// TIA Portal project "Winda2.2" (V15.1)

(* hardware
DEVICE "S7-1200 station_1"  S7-1200 Station
   slot 0: "Rack_0"  S7-1200 Rack  Rack  V1.0
   slot 1: "PLC_1"  CPU 1212C AC/DC/Rly  6ES7 212-1BD30-0XB0  V2.2
DEVICE "HMI_1"  KTP600 Basic color PN
   slot 0: "HMI_1"  KTP600 Basic color PN  6AV6 647-0AD11-3AX0  12.0.0.0
   slot 1: "HMI_RT_1"  KTP600 Basic color PN  6AV6 647-0AD11-3AX0  12.0.0.0
   slot 5: "HMI_1.IE_CP_1"  PROFINET Interface  12.0.0.0
      slot 1: "PROFINET Interface_1"  PROFINET Interface
         slot 1: "Port_1"  Port
*)

// ===== PLC "PLC_1"  CPU 1212C AC/DC/Rly =====

VAR_GLOBAL   // PLC tag table "Default tag table"
   "Btn_0_floor_out" AT %M0.0 : Bool;
   "Btn_1_floor_out" AT %M0.1 : Bool;
   "Btn_2_floor_out" AT %M0.2 : Bool;
   "Btn_3_floor_out" AT %M0.3 : Bool;
   "Btn_4_floor_out" AT %M0.4 : Bool;
   "Btn_5_floor_out" AT %M0.5 : Bool;
   "Btn_6_floor_out" AT %M0.6 : Bool;
   "Btn_7_floor_out" AT %M0.7 : Bool;
   "Btn_8_floor_out" AT %M1.0 : Bool;
   "Btn_9_floor_out" AT %M1.1 : Bool;
   "Btn_10_floor_out" AT %M1.2 : Bool;
   "Btn_0_floor_in" AT %M1.3 : Bool;
   "Btn_1_floor_in" AT %M1.4 : Bool;
   "Btn_2_floor_in" AT %M1.5 : Bool;
   "Btn_3_floor_in" AT %M1.6 : Bool;
   "Btn_4_floor_in" AT %M1.7 : Bool;
   "Btn_5_floor_in" AT %M2.0 : Bool;
   "Btn_6_floor_in" AT %M2.1 : Bool;
   "Btn_7_floor_in" AT %M2.2 : Bool;
   "Btn_8_floor_in" AT %M2.3 : Bool;
   "Btn_9_floor_in" AT %M2.4 : Bool;
   "Btn_10_floor_in" AT %M2.5 : Bool;
   "Btn_emergency" AT %M2.6 : Bool;
   "Btn_open_door" AT %M2.7 : Bool;
   "Btn_close_door" AT %M3.0 : Bool;
   "DO_open_door" AT %M3.1 : Bool;
   "DO_close_door" AT %M3.2 : Bool;
   "DO_move_lift_up" AT %M3.3 : Bool;
   "DO_move_lift_down" AT %M3.4 : Bool;
   "DO_motor_brake" AT %M3.5 : Bool;
   "MoveTimerIN" AT %M3.6 : Bool;
   "DoorTimerIN" AT %M3.7 : Bool;
   "MoveTimerStoppingIN" AT %M4.0 : Bool;
   "Clock_Byte" AT %MB100 : Byte;
   "Clock_10Hz" AT %M100.0 : Bool;
   "Clock_5Hz" AT %M100.1 : Bool;
   "Clock_2.5Hz" AT %M100.2 : Bool;
   "Clock_2Hz" AT %M100.3 : Bool;
   "Clock_1.25Hz" AT %M100.4 : Bool;
   "Clock_1Hz" AT %M100.5 : Bool;
   "Clock_0.625Hz" AT %M100.6 : Bool;
   "Clock_0.5Hz" AT %M100.7 : Bool;
   "HMIElevatorPosition" AT %MW7 : Int;
   "HMIReq_0" AT %M4.1 : Bool;
   "HMIReq_1" AT %M4.2 : Bool;
   "HMIReq_2" AT %M4.3 : Bool;
   "HMIReq_3" AT %M4.4 : Bool;
   "HMIReq_4" AT %M4.5 : Bool;
   "HMIReq_5" AT %M4.6 : Bool;
   "HMIReq_6" AT %M4.7 : Bool;
   "HMIReq_7" AT %M5.0 : Bool;
   "HMIReq_8" AT %M5.1 : Bool;
   "HMIReq_9" AT %M5.2 : Bool;
   "HMIReq_10" AT %M5.3 : Bool;
   "HMIDoorPosition" AT %MW9 : Int;
   "P1" AT %M5.4 : Bool;
   "P2" AT %M5.5 : Bool;
   "P3" AT %M5.6 : Bool;
   "P4" AT %M5.7 : Bool;
   "P5" AT %M6.0 : Bool;
   "P6" AT %M6.1 : Bool;
   "P7" AT %M6.2 : Bool;
   "P8" AT %M6.3 : Bool;
   "N1" AT %M6.4 : Bool;
END_VAR

VAR_GLOBAL CONSTANT   // PLC tag table "Default tag table"
   "ES_IDLE" : Int := 0;
   "ES_DOOR_OPEN" : Int := 1;
   "ES_MOVING_UP" : Int := 2;
   "ES_MOVING_DOWN" : Int := 3;
   "ES_STOPPING" : Int := 4;
END_VAR

DATA_BLOCK "Elevator"   // DB2
{ S7_Optimized_Access := 'TRUE' }
VERSION : 0.1
   VAR
      Requests : Array[0..10] of Bool;
      state : Int;
      currentFloor : Int;
      targetFloor : Int;
      DoorState : Int := 2;
      DoorTimerPT : Time := T#3ms;
      MoveTimerPT : Time := T#2s;
      MoveTimerStoppingPT : Time := T#4s;
      BeforeEmergancyState : Int;
      DoorTimerWasON : Bool;
      MoveTimerWasON : Bool;
      MoveTimerStoppingWasON : Bool;
      DoorTimerET : Time;
      MoveTimerET : Time;
      MoveTimerStoppingET : Time;
      MotorState : Bool;
   END_VAR
BEGIN
END_DATA_BLOCK

DATA_BLOCK "HMIsim_DB"   // DB5
{ S7_Optimized_Access := 'TRUE' }
VERSION : 0.1
// stored: InstanceOfName HMIsim
"HMIsim"
BEGIN
END_DATA_BLOCK

DATA_BLOCK "UpdateDoorPosition_DB"   // DB6
{ S7_Optimized_Access := 'TRUE' }
VERSION : 0.1
// stored: InstanceOfName UpdateDoorPosition
"UpdateDoorPosition"
BEGIN
END_DATA_BLOCK

// folder: System blocks/Program resources

DATA_BLOCK "DoorTimer"   // DB1
{ S7_Optimized_Access := 'TRUE' }
AUTHOR : Simatic
FAMILY : IEC
NAME : IEC_TMR
VERSION : 1.0
// stored: InstanceOfName IEC_TIMER
"IEC_TIMER"
BEGIN
END_DATA_BLOCK

DATA_BLOCK "MoveTimer"   // DB3
{ S7_Optimized_Access := 'TRUE' }
AUTHOR : Simatic
FAMILY : IEC
NAME : IEC_TMR
VERSION : 1.0
// stored: InstanceOfName IEC_TIMER
"IEC_TIMER"
BEGIN
END_DATA_BLOCK

DATA_BLOCK "MoveTimerStopping"   // DB4
{ S7_Optimized_Access := 'TRUE' }
AUTHOR : Simatic
FAMILY : IEC
NAME : IEC_TMR
VERSION : 1.0
// stored: InstanceOfName IEC_TIMER
"IEC_TIMER"
BEGIN
END_DATA_BLOCK

// folder: (top level)

FUNCTION_BLOCK "HMIsim"   // FB1, LAD
{ S7_Optimized_Access := 'TRUE' }
VERSION : 0.1
   VAR_INPUT
      StartTravel : Bool;
      TargetFloorIndex : Int;
   END_VAR
   VAR_OUTPUT
      ElevatorPos : Int;
   END_VAR
   VAR_TEMP
      direction : Int;
      CurrentStartPos : Int;
      NextFloorPos : Int;
      temp1 : Int;
      ET_int : Int;
      PositionProgress : Real;
      ET_R : Real;
      temp2 : Real;
   END_VAR
   VAR CONSTANT
      StepDistance : Int := 21;
      TotalRange : Int := 210;
      TotalSteps : Int := 10;
   END_VAR
   VAR_TEMP   // added for the SCL form of the ladder/FBD networks
      _w1 : Bool;
      _w2 : Bool;
      _w3 : Bool;
      _w4 : Bool;
   END_VAR
BEGIN

REGION Network 1
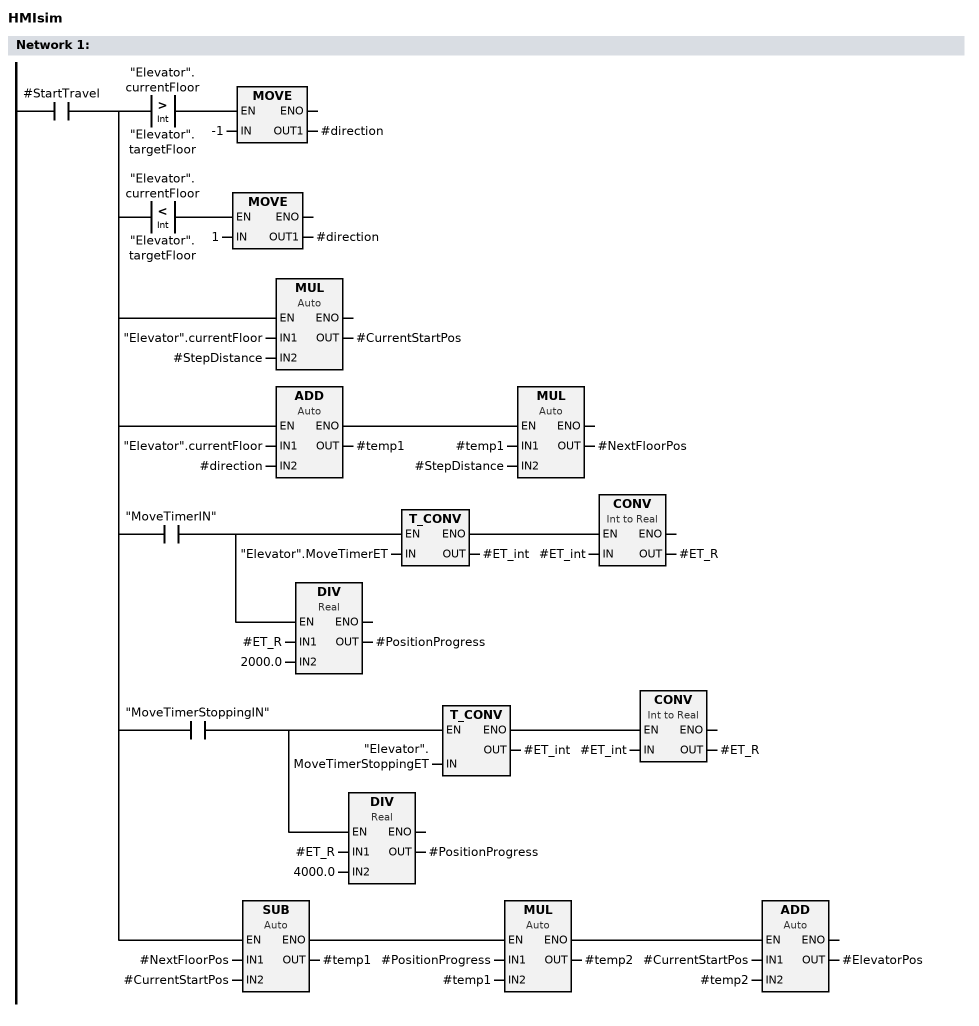
   // ENO of a box is taken as its EN; it also drops when the box reports an error
   IF #StartTravel AND ("Elevator".currentFloor > "Elevator".targetFloor) THEN #direction := -1; END_IF;
   IF #StartTravel AND ("Elevator".currentFloor < "Elevator".targetFloor) THEN #direction := 1; END_IF;
   IF #StartTravel THEN
       #CurrentStartPos := "Elevator".currentFloor * #StepDistance;
       #temp1 := "Elevator".currentFloor + #direction;
       #NextFloorPos := #temp1 * #StepDistance;
   END_IF;
   #_w1 := #StartTravel AND "MoveTimerIN";
   #_w2 := #StartTravel AND "MoveTimerIN";
   IF #_w2 THEN
       #ET_int := T_CONV(IN := "Elevator".MoveTimerET);
       #ET_R := INT_TO_REAL(#ET_int);
   END_IF;
   IF #_w1 THEN #PositionProgress := #ET_R / 2000.0; END_IF;
   #_w3 := #StartTravel AND "MoveTimerStoppingIN";
   #_w4 := #StartTravel AND "MoveTimerStoppingIN";
   IF #_w4 THEN
       #ET_int := T_CONV(IN := "Elevator".MoveTimerStoppingET);
       #ET_R := INT_TO_REAL(#ET_int);
   END_IF;
   IF #_w3 THEN #PositionProgress := #ET_R / 4000.0; END_IF;
   IF #StartTravel THEN
       #temp1 := #NextFloorPos - #CurrentStartPos;
       #temp2 := #PositionProgress * #temp1;
       #ElevatorPos := #CurrentStartPos + #temp2;
   END_IF;
END_REGION
END_FUNCTION_BLOCK

FUNCTION_BLOCK "UpdateDoorPosition"   // FB2, LAD
{ S7_Optimized_Access := 'TRUE' }
VERSION : 0.1
   VAR_INPUT
      TimeElapsed : Time;
   END_VAR
   VAR
      DoorRange : Real := 30.0;
      DoorTimeTotal : Time := T#3s;
   END_VAR
   VAR_TEMP
      TimeFraction : Real;
      Temp_1 : Int;
      Temp_2 : Int;
      Temp_3 : Real;
   END_VAR
BEGIN

REGION Network 1
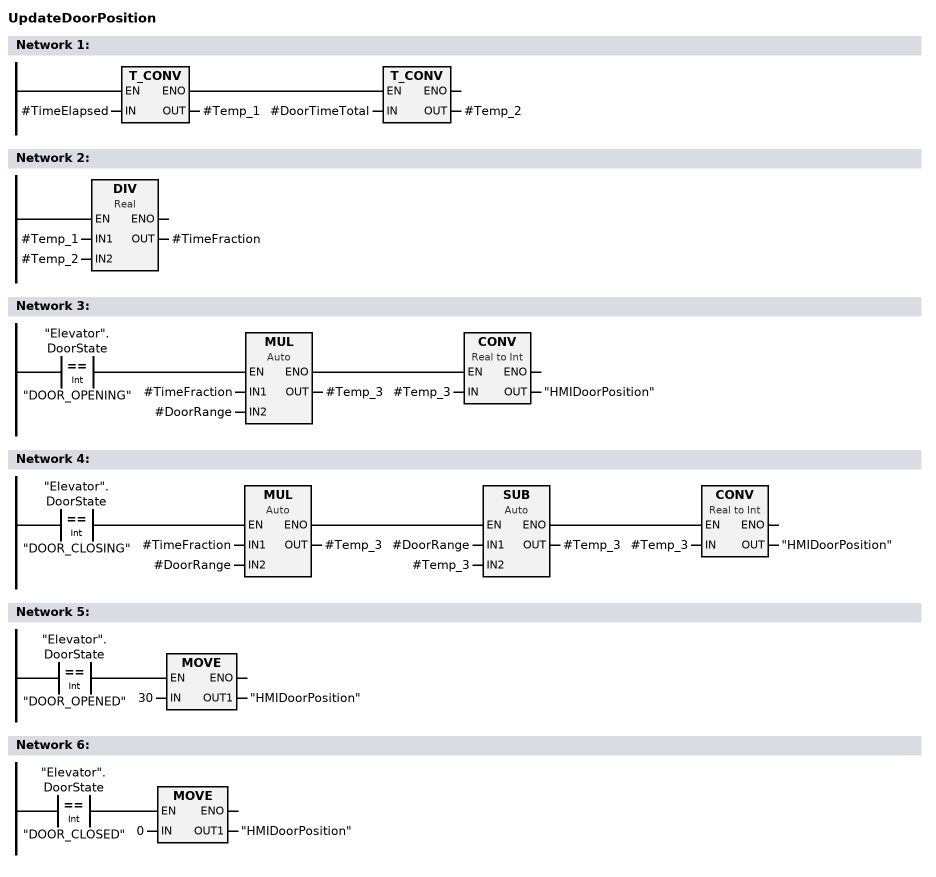
   // ENO of a box is taken as its EN; it also drops when the box reports an error
   #Temp_1 := T_CONV(IN := #TimeElapsed);
   #Temp_2 := T_CONV(IN := #DoorTimeTotal);
END_REGION

REGION Network 2
   RUNG wire#powerrail
      { S7_Templates := "SrcType := Real" } Div(in1 := #Temp_1, in2 := #Temp_2, out => #TimeFraction)
   END_RUNG
   // the same network as SCL:
   #TimeFraction := #Temp_1 / #Temp_2;
END_REGION

REGION Network 3
   RUNG wire#powerrail
      { S7_Templates := "SrcType := Int" } EQ_Contact(in1 := "Elevator".DoorState, in2 := "DOOR_OPENING")
      Mul(in1 := #TimeFraction, in2 := #DoorRange, out => #Temp_3)
      { S7_Templates := "[SrcType := Real, DestType := Int]" } Convert(in := #Temp_3, out => "HMIDoorPosition")
   END_RUNG
   // the same network as SCL:
   IF "Elevator".DoorState = "DOOR_OPENING" THEN
       #Temp_3 := #TimeFraction * #DoorRange;
       "HMIDoorPosition" := REAL_TO_INT(#Temp_3);
   END_IF;
END_REGION

REGION Network 4
   RUNG wire#powerrail
      { S7_Templates := "SrcType := Int" } EQ_Contact(in1 := "Elevator".DoorState, in2 := "DOOR_CLOSING")
      Mul(in1 := #TimeFraction, in2 := #DoorRange, out => #Temp_3)
      Sub(in1 := #DoorRange, in2 := #Temp_3, out => #Temp_3)
      { S7_Templates := "[SrcType := Real, DestType := Int]" } Convert(in := #Temp_3, out => "HMIDoorPosition")
   END_RUNG
   // the same network as SCL:
   IF "Elevator".DoorState = "DOOR_CLOSING" THEN
       #Temp_3 := #TimeFraction * #DoorRange;
       #Temp_3 := #DoorRange - #Temp_3;
       "HMIDoorPosition" := REAL_TO_INT(#Temp_3);
   END_IF;
END_REGION

REGION Network 5
   RUNG wire#powerrail
      { S7_Templates := "SrcType := Int" } EQ_Contact(in1 := "Elevator".DoorState, in2 := "DOOR_OPENED")
      Move(in := 30, out1 => "HMIDoorPosition")
   END_RUNG
   // the same network as SCL:
   IF "Elevator".DoorState = "DOOR_OPENED" THEN "HMIDoorPosition" := 30; END_IF;
END_REGION

REGION Network 6
   RUNG wire#powerrail
      { S7_Templates := "SrcType := Int" } EQ_Contact(in1 := "Elevator".DoorState, in2 := "DOOR_CLOSED")
      Move(in := 0, out1 => "HMIDoorPosition")
   END_RUNG
   // the same network as SCL:
   IF "Elevator".DoorState = "DOOR_CLOSED" THEN "HMIDoorPosition" := 0; END_IF;
END_REGION
END_FUNCTION_BLOCK

FUNCTION "GetPendingRequests" : Void   // FC2, LAD
{ S7_Optimized_Access := 'TRUE' }
VERSION : 0.1
   VAR_INPUT
      Btn_0_floor_out : Bool;
      Btn_1_floor_out : Bool;
      Btn_2_floor_out : Bool;
      Btn_3_floor_out : Bool;
      Btn_4_floor_out : Bool;
      Btn_5_floor_out : Bool;
      Btn_6_floor_out : Bool;
      Btn_7_floor_out : Bool;
      Btn_8_floor_out : Bool;
      Btn_9_floor_out : Bool;
      Btn_10_floor_out : Bool;
      Btn_0_floor_in : Bool;
      Btn_1_floor_in : Bool;
      Btn_2_floor_in : Bool;
      Btn_3_floor_in : Bool;
      Btn_4_floor_in : Bool;
      Btn_5_floor_in : Bool;
      Btn_6_floor_in : Bool;
      Btn_7_floor_in : Bool;
      Btn_8_floor_in : Bool;
      Btn_9_floor_in : Bool;
      Btn_10_floor_in : Bool;
   END_VAR
   VAR_OUTPUT
      requests : Array[0..10] of Bool;
   END_VAR
BEGIN

REGION Network 1
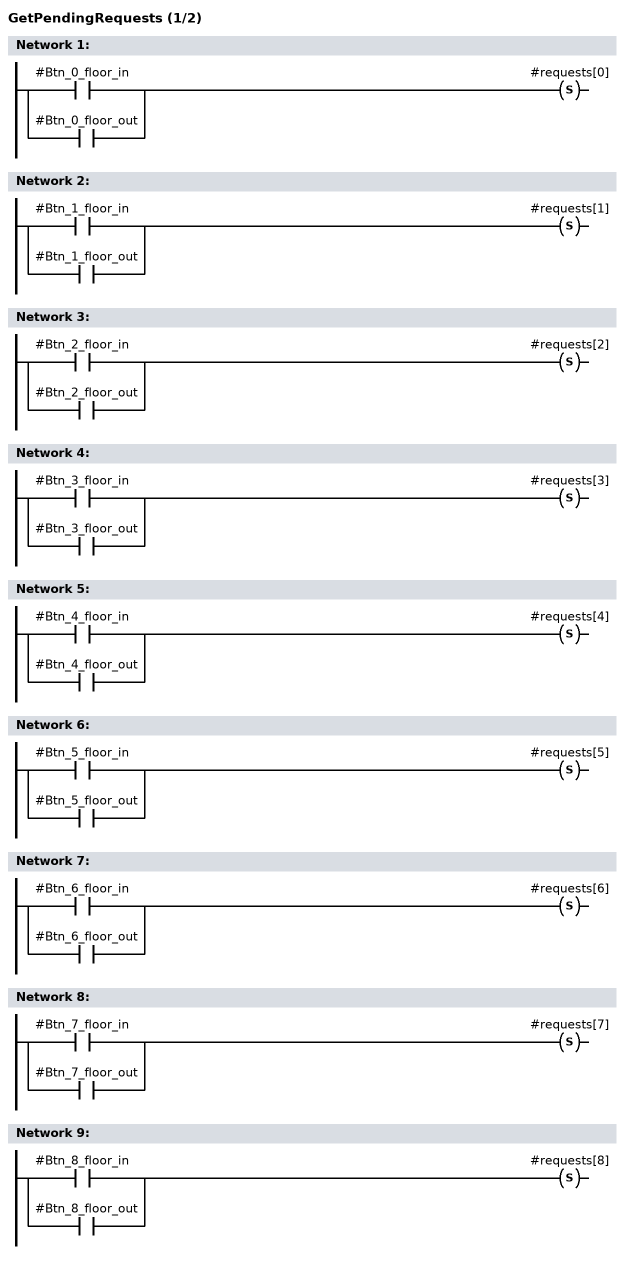
   RUNG wire#powerrail
      Contact( #Btn_0_floor_in )
      wire#w1
      S_Coil( #requests[0] )
   END_RUNG
   RUNG wire#powerrail
      Contact( #Btn_0_floor_out )
   END_RUNG wire#w1
   // the same network as SCL:
   IF #Btn_0_floor_in OR #Btn_0_floor_out THEN #requests[0] := TRUE; END_IF;
END_REGION

REGION Network 2
   RUNG wire#powerrail
      Contact( #Btn_1_floor_in )
      wire#w1
      S_Coil( #requests[1] )
   END_RUNG
   RUNG wire#powerrail
      Contact( #Btn_1_floor_out )
   END_RUNG wire#w1
   // the same network as SCL:
   IF #Btn_1_floor_in OR #Btn_1_floor_out THEN #requests[1] := TRUE; END_IF;
END_REGION

REGION Network 3
   RUNG wire#powerrail
      Contact( #Btn_2_floor_in )
      wire#w1
      S_Coil( #requests[2] )
   END_RUNG
   RUNG wire#powerrail
      Contact( #Btn_2_floor_out )
   END_RUNG wire#w1
   // the same network as SCL:
   IF #Btn_2_floor_in OR #Btn_2_floor_out THEN #requests[2] := TRUE; END_IF;
END_REGION

REGION Network 4
   RUNG wire#powerrail
      Contact( #Btn_3_floor_in )
      wire#w1
      S_Coil( #requests[3] )
   END_RUNG
   RUNG wire#powerrail
      Contact( #Btn_3_floor_out )
   END_RUNG wire#w1
   // the same network as SCL:
   IF #Btn_3_floor_in OR #Btn_3_floor_out THEN #requests[3] := TRUE; END_IF;
END_REGION

REGION Network 5
   RUNG wire#powerrail
      Contact( #Btn_4_floor_in )
      wire#w1
      S_Coil( #requests[4] )
   END_RUNG
   RUNG wire#powerrail
      Contact( #Btn_4_floor_out )
   END_RUNG wire#w1
   // the same network as SCL:
   IF #Btn_4_floor_in OR #Btn_4_floor_out THEN #requests[4] := TRUE; END_IF;
END_REGION

REGION Network 6
   RUNG wire#powerrail
      Contact( #Btn_5_floor_in )
      wire#w1
      S_Coil( #requests[5] )
   END_RUNG
   RUNG wire#powerrail
      Contact( #Btn_5_floor_out )
   END_RUNG wire#w1
   // the same network as SCL:
   IF #Btn_5_floor_in OR #Btn_5_floor_out THEN #requests[5] := TRUE; END_IF;
END_REGION

REGION Network 7
   RUNG wire#powerrail
      Contact( #Btn_6_floor_in )
      wire#w1
      S_Coil( #requests[6] )
   END_RUNG
   RUNG wire#powerrail
      Contact( #Btn_6_floor_out )
   END_RUNG wire#w1
   // the same network as SCL:
   IF #Btn_6_floor_in OR #Btn_6_floor_out THEN #requests[6] := TRUE; END_IF;
END_REGION

REGION Network 8
   RUNG wire#powerrail
      Contact( #Btn_7_floor_in )
      wire#w1
      S_Coil( #requests[7] )
   END_RUNG
   RUNG wire#powerrail
      Contact( #Btn_7_floor_out )
   END_RUNG wire#w1
   // the same network as SCL:
   IF #Btn_7_floor_in OR #Btn_7_floor_out THEN #requests[7] := TRUE; END_IF;
END_REGION

REGION Network 9
   RUNG wire#powerrail
      Contact( #Btn_8_floor_in )
      wire#w1
      S_Coil( #requests[8] )
   END_RUNG
   RUNG wire#powerrail
      Contact( #Btn_8_floor_out )
   END_RUNG wire#w1
   // the same network as SCL:
   IF #Btn_8_floor_in OR #Btn_8_floor_out THEN #requests[8] := TRUE; END_IF;
END_REGION

REGION Network 10
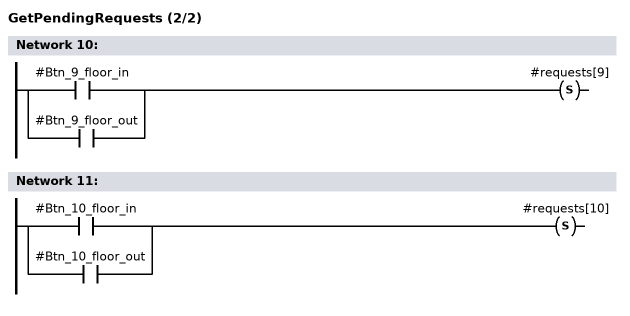
   RUNG wire#powerrail
      Contact( #Btn_9_floor_in )
      wire#w1
      S_Coil( #requests[9] )
   END_RUNG
   RUNG wire#powerrail
      Contact( #Btn_9_floor_out )
   END_RUNG wire#w1
   // the same network as SCL:
   IF #Btn_9_floor_in OR #Btn_9_floor_out THEN #requests[9] := TRUE; END_IF;
END_REGION

REGION Network 11
   RUNG wire#powerrail
      Contact( #Btn_10_floor_in )
      wire#w1
      S_Coil( #requests[10] )
   END_RUNG
   RUNG wire#powerrail
      Contact( #Btn_10_floor_out )
   END_RUNG wire#w1
   // the same network as SCL:
   IF #Btn_10_floor_in OR #Btn_10_floor_out THEN #requests[10] := TRUE; END_IF;
END_REGION
END_FUNCTION

FUNCTION "RequestExists" : Bool   // FC3, LAD
{ S7_Optimized_Access := 'TRUE' }
VERSION : 0.1
BEGIN

REGION Network 1
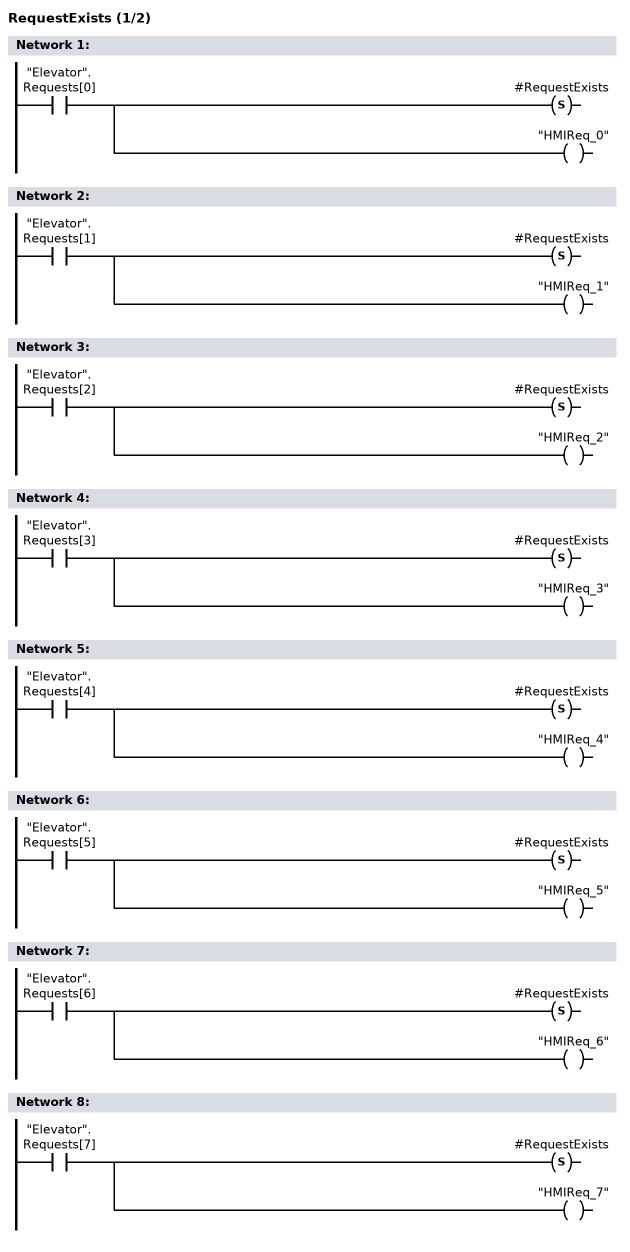
   RUNG wire#powerrail
      Contact( "Elevator".Requests[0] )
      wire#w1
      S_Coil( #RequestExists )
   END_RUNG
   RUNG wire#w1
      Coil( "HMIReq_0" )
   END_RUNG
   // the same network as SCL:
   IF "Elevator".Requests[0] THEN #RequestExists := TRUE; END_IF;
   "HMIReq_0" := "Elevator".Requests[0];
END_REGION

REGION Network 2
   RUNG wire#powerrail
      Contact( "Elevator".Requests[1] )
      wire#w1
      S_Coil( #RequestExists )
   END_RUNG
   RUNG wire#w1
      Coil( "HMIReq_1" )
   END_RUNG
   // the same network as SCL:
   IF "Elevator".Requests[1] THEN #RequestExists := TRUE; END_IF;
   "HMIReq_1" := "Elevator".Requests[1];
END_REGION

REGION Network 3
   RUNG wire#powerrail
      Contact( "Elevator".Requests[2] )
      wire#w1
      S_Coil( #RequestExists )
   END_RUNG
   RUNG wire#w1
      Coil( "HMIReq_2" )
   END_RUNG
   // the same network as SCL:
   IF "Elevator".Requests[2] THEN #RequestExists := TRUE; END_IF;
   "HMIReq_2" := "Elevator".Requests[2];
END_REGION

REGION Network 4
   RUNG wire#powerrail
      Contact( "Elevator".Requests[3] )
      wire#w1
      S_Coil( #RequestExists )
   END_RUNG
   RUNG wire#w1
      Coil( "HMIReq_3" )
   END_RUNG
   // the same network as SCL:
   IF "Elevator".Requests[3] THEN #RequestExists := TRUE; END_IF;
   "HMIReq_3" := "Elevator".Requests[3];
END_REGION

REGION Network 5
   RUNG wire#powerrail
      Contact( "Elevator".Requests[4] )
      wire#w1
      S_Coil( #RequestExists )
   END_RUNG
   RUNG wire#w1
      Coil( "HMIReq_4" )
   END_RUNG
   // the same network as SCL:
   IF "Elevator".Requests[4] THEN #RequestExists := TRUE; END_IF;
   "HMIReq_4" := "Elevator".Requests[4];
END_REGION

REGION Network 6
   RUNG wire#powerrail
      Contact( "Elevator".Requests[5] )
      wire#w1
      S_Coil( #RequestExists )
   END_RUNG
   RUNG wire#w1
      Coil( "HMIReq_5" )
   END_RUNG
   // the same network as SCL:
   IF "Elevator".Requests[5] THEN #RequestExists := TRUE; END_IF;
   "HMIReq_5" := "Elevator".Requests[5];
END_REGION

REGION Network 7
   RUNG wire#powerrail
      Contact( "Elevator".Requests[6] )
      wire#w1
      S_Coil( #RequestExists )
   END_RUNG
   RUNG wire#w1
      Coil( "HMIReq_6" )
   END_RUNG
   // the same network as SCL:
   IF "Elevator".Requests[6] THEN #RequestExists := TRUE; END_IF;
   "HMIReq_6" := "Elevator".Requests[6];
END_REGION

REGION Network 8
   RUNG wire#powerrail
      Contact( "Elevator".Requests[7] )
      wire#w1
      S_Coil( #RequestExists )
   END_RUNG
   RUNG wire#w1
      Coil( "HMIReq_7" )
   END_RUNG
   // the same network as SCL:
   IF "Elevator".Requests[7] THEN #RequestExists := TRUE; END_IF;
   "HMIReq_7" := "Elevator".Requests[7];
END_REGION

REGION Network 9
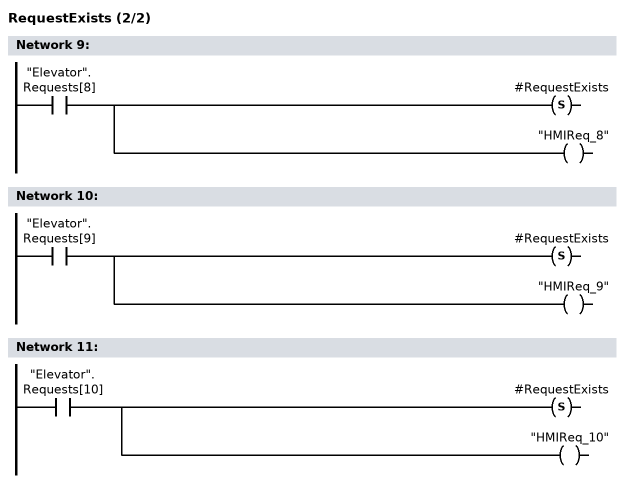
   RUNG wire#powerrail
      Contact( "Elevator".Requests[8] )
      wire#w1
      S_Coil( #RequestExists )
   END_RUNG
   RUNG wire#w1
      Coil( "HMIReq_8" )
   END_RUNG
   // the same network as SCL:
   IF "Elevator".Requests[8] THEN #RequestExists := TRUE; END_IF;
   "HMIReq_8" := "Elevator".Requests[8];
END_REGION

REGION Network 10
   RUNG wire#powerrail
      Contact( "Elevator".Requests[9] )
      wire#w1
      S_Coil( #RequestExists )
   END_RUNG
   RUNG wire#w1
      Coil( "HMIReq_9" )
   END_RUNG
   // the same network as SCL:
   IF "Elevator".Requests[9] THEN #RequestExists := TRUE; END_IF;
   "HMIReq_9" := "Elevator".Requests[9];
END_REGION

REGION Network 11
   RUNG wire#powerrail
      Contact( "Elevator".Requests[10] )
      wire#w1
      S_Coil( #RequestExists )
   END_RUNG
   RUNG wire#w1
      Coil( "HMIReq_10" )
   END_RUNG
   // the same network as SCL:
   IF "Elevator".Requests[10] THEN #RequestExists := TRUE; END_IF;
   "HMIReq_10" := "Elevator".Requests[10];
END_REGION
END_FUNCTION

FUNCTION "GetNextTarget" : Int   // FC4, LAD
{ S7_Optimized_Access := 'TRUE' }
VERSION : 0.1
   VAR_INPUT
      current : Int;
      req : Array[0..10] of Bool;
   END_VAR
   VAR_TEMP
      minDiff : Int;
      diff : Int;
      temp1 : Int;
      temp2 : Int;
      nextTarget : Int;
   END_VAR
   VAR_TEMP   // added for the SCL form of the ladder/FBD networks
      _w1 : Bool;
   END_VAR
BEGIN

REGION Network 1
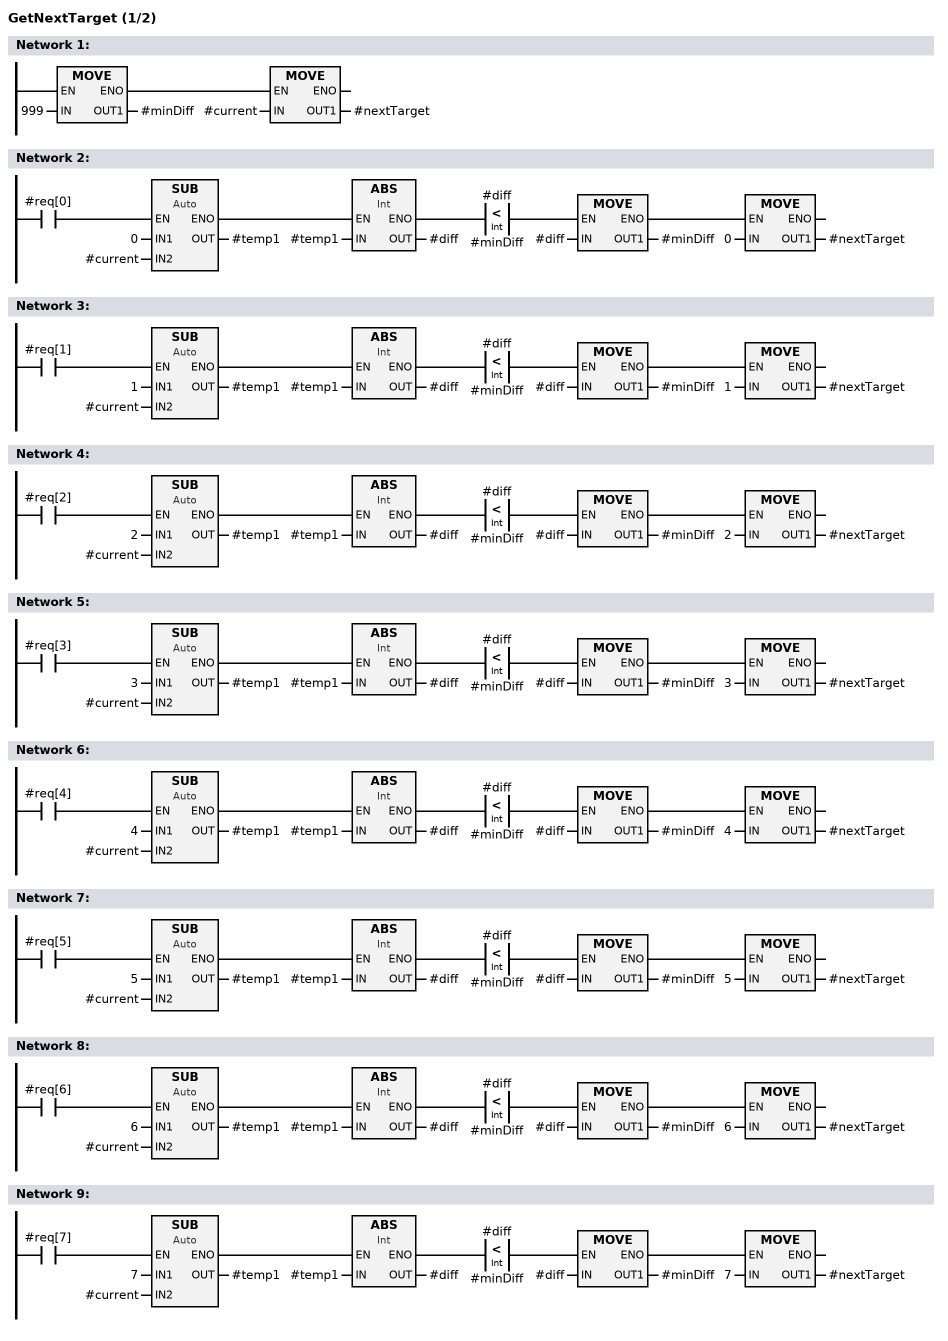
   RUNG wire#powerrail
      { S7_GenerateENO := "TRUE" } Move(in := 999, out1 => #minDiff)
      { S7_GenerateENO := "TRUE" } Move(in := #current, out1 => #nextTarget)
   END_RUNG
   // the same network as SCL:
   // ENO of a box is taken as its EN; it also drops when the box reports an error
   #minDiff := 999;
   #nextTarget := #current;
END_REGION

REGION Network 2
   RUNG wire#powerrail
      Contact( #req[0] )
      { S7_GenerateENO := "TRUE" } Sub(in1 := 0, in2 := #current, out => #temp1)
      { S7_Templates := "SrcType := Int"; S7_GenerateENO := "TRUE" } Abs(in := #temp1, out => #diff)
      { S7_Templates := "SrcType := Int" } LT_Contact(in1 := #diff, in2 := #minDiff)
      { S7_GenerateENO := "TRUE" } Move(in := #diff, out1 => #minDiff)
      { S7_GenerateENO := "TRUE" } Move(in := 0, out1 => #nextTarget)
   END_RUNG
   // the same network as SCL:
   // ENO of a box is taken as its EN; it also drops when the box reports an error
   IF #req[0] THEN
       #temp1 := 0 - #current;
       #diff := ABS(#temp1);
   END_IF;
   #_w1 := #req[0] AND (#diff < #minDiff);
   IF #_w1 THEN
       #minDiff := #diff;
       #nextTarget := 0;
   END_IF;
END_REGION

REGION Network 3
   RUNG wire#powerrail
      Contact( #req[1] )
      { S7_GenerateENO := "TRUE" } Sub(in1 := 1, in2 := #current, out => #temp1)
      { S7_Templates := "SrcType := Int"; S7_GenerateENO := "TRUE" } Abs(in := #temp1, out => #diff)
      { S7_Templates := "SrcType := Int" } LT_Contact(in1 := #diff, in2 := #minDiff)
      { S7_GenerateENO := "TRUE" } Move(in := #diff, out1 => #minDiff)
      { S7_GenerateENO := "TRUE" } Move(in := 1, out1 => #nextTarget)
   END_RUNG
   // the same network as SCL:
   // ENO of a box is taken as its EN; it also drops when the box reports an error
   IF #req[1] THEN
       #temp1 := 1 - #current;
       #diff := ABS(#temp1);
   END_IF;
   #_w1 := #req[1] AND (#diff < #minDiff);
   IF #_w1 THEN
       #minDiff := #diff;
       #nextTarget := 1;
   END_IF;
END_REGION

REGION Network 4
   RUNG wire#powerrail
      Contact( #req[2] )
      { S7_GenerateENO := "TRUE" } Sub(in1 := 2, in2 := #current, out => #temp1)
      { S7_Templates := "SrcType := Int"; S7_GenerateENO := "TRUE" } Abs(in := #temp1, out => #diff)
      { S7_Templates := "SrcType := Int" } LT_Contact(in1 := #diff, in2 := #minDiff)
      { S7_GenerateENO := "TRUE" } Move(in := #diff, out1 => #minDiff)
      { S7_GenerateENO := "TRUE" } Move(in := 2, out1 => #nextTarget)
   END_RUNG
   // the same network as SCL:
   // ENO of a box is taken as its EN; it also drops when the box reports an error
   IF #req[2] THEN
       #temp1 := 2 - #current;
       #diff := ABS(#temp1);
   END_IF;
   #_w1 := #req[2] AND (#diff < #minDiff);
   IF #_w1 THEN
       #minDiff := #diff;
       #nextTarget := 2;
   END_IF;
END_REGION

REGION Network 5
   RUNG wire#powerrail
      Contact( #req[3] )
      { S7_GenerateENO := "TRUE" } Sub(in1 := 3, in2 := #current, out => #temp1)
      { S7_Templates := "SrcType := Int"; S7_GenerateENO := "TRUE" } Abs(in := #temp1, out => #diff)
      { S7_Templates := "SrcType := Int" } LT_Contact(in1 := #diff, in2 := #minDiff)
      { S7_GenerateENO := "TRUE" } Move(in := #diff, out1 => #minDiff)
      { S7_GenerateENO := "TRUE" } Move(in := 3, out1 => #nextTarget)
   END_RUNG
   // the same network as SCL:
   // ENO of a box is taken as its EN; it also drops when the box reports an error
   IF #req[3] THEN
       #temp1 := 3 - #current;
       #diff := ABS(#temp1);
   END_IF;
   #_w1 := #req[3] AND (#diff < #minDiff);
   IF #_w1 THEN
       #minDiff := #diff;
       #nextTarget := 3;
   END_IF;
END_REGION

REGION Network 6
   RUNG wire#powerrail
      Contact( #req[4] )
      { S7_GenerateENO := "TRUE" } Sub(in1 := 4, in2 := #current, out => #temp1)
      { S7_Templates := "SrcType := Int"; S7_GenerateENO := "TRUE" } Abs(in := #temp1, out => #diff)
      { S7_Templates := "SrcType := Int" } LT_Contact(in1 := #diff, in2 := #minDiff)
      { S7_GenerateENO := "TRUE" } Move(in := #diff, out1 => #minDiff)
      { S7_GenerateENO := "TRUE" } Move(in := 4, out1 => #nextTarget)
   END_RUNG
   // the same network as SCL:
   // ENO of a box is taken as its EN; it also drops when the box reports an error
   IF #req[4] THEN
       #temp1 := 4 - #current;
       #diff := ABS(#temp1);
   END_IF;
   #_w1 := #req[4] AND (#diff < #minDiff);
   IF #_w1 THEN
       #minDiff := #diff;
       #nextTarget := 4;
   END_IF;
END_REGION

REGION Network 7
   RUNG wire#powerrail
      Contact( #req[5] )
      { S7_GenerateENO := "TRUE" } Sub(in1 := 5, in2 := #current, out => #temp1)
      { S7_Templates := "SrcType := Int"; S7_GenerateENO := "TRUE" } Abs(in := #temp1, out => #diff)
      { S7_Templates := "SrcType := Int" } LT_Contact(in1 := #diff, in2 := #minDiff)
      { S7_GenerateENO := "TRUE" } Move(in := #diff, out1 => #minDiff)
      { S7_GenerateENO := "TRUE" } Move(in := 5, out1 => #nextTarget)
   END_RUNG
   // the same network as SCL:
   // ENO of a box is taken as its EN; it also drops when the box reports an error
   IF #req[5] THEN
       #temp1 := 5 - #current;
       #diff := ABS(#temp1);
   END_IF;
   #_w1 := #req[5] AND (#diff < #minDiff);
   IF #_w1 THEN
       #minDiff := #diff;
       #nextTarget := 5;
   END_IF;
END_REGION

REGION Network 8
   RUNG wire#powerrail
      Contact( #req[6] )
      { S7_GenerateENO := "TRUE" } Sub(in1 := 6, in2 := #current, out => #temp1)
      { S7_Templates := "SrcType := Int"; S7_GenerateENO := "TRUE" } Abs(in := #temp1, out => #diff)
      { S7_Templates := "SrcType := Int" } LT_Contact(in1 := #diff, in2 := #minDiff)
      { S7_GenerateENO := "TRUE" } Move(in := #diff, out1 => #minDiff)
      { S7_GenerateENO := "TRUE" } Move(in := 6, out1 => #nextTarget)
   END_RUNG
   // the same network as SCL:
   // ENO of a box is taken as its EN; it also drops when the box reports an error
   IF #req[6] THEN
       #temp1 := 6 - #current;
       #diff := ABS(#temp1);
   END_IF;
   #_w1 := #req[6] AND (#diff < #minDiff);
   IF #_w1 THEN
       #minDiff := #diff;
       #nextTarget := 6;
   END_IF;
END_REGION

REGION Network 9
   RUNG wire#powerrail
      Contact( #req[7] )
      { S7_GenerateENO := "TRUE" } Sub(in1 := 7, in2 := #current, out => #temp1)
      { S7_Templates := "SrcType := Int"; S7_GenerateENO := "TRUE" } Abs(in := #temp1, out => #diff)
      { S7_Templates := "SrcType := Int" } LT_Contact(in1 := #diff, in2 := #minDiff)
      { S7_GenerateENO := "TRUE" } Move(in := #diff, out1 => #minDiff)
      { S7_GenerateENO := "TRUE" } Move(in := 7, out1 => #nextTarget)
   END_RUNG
   // the same network as SCL:
   // ENO of a box is taken as its EN; it also drops when the box reports an error
   IF #req[7] THEN
       #temp1 := 7 - #current;
       #diff := ABS(#temp1);
   END_IF;
   #_w1 := #req[7] AND (#diff < #minDiff);
   IF #_w1 THEN
       #minDiff := #diff;
       #nextTarget := 7;
   END_IF;
END_REGION

REGION Network 10
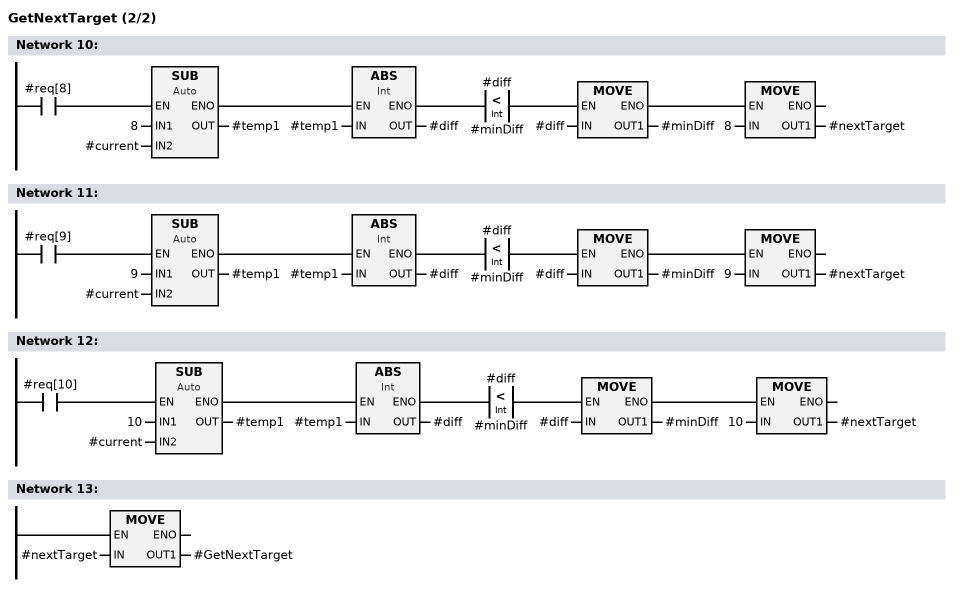
   RUNG wire#powerrail
      Contact( #req[8] )
      { S7_GenerateENO := "TRUE" } Sub(in1 := 8, in2 := #current, out => #temp1)
      { S7_Templates := "SrcType := Int"; S7_GenerateENO := "TRUE" } Abs(in := #temp1, out => #diff)
      { S7_Templates := "SrcType := Int" } LT_Contact(in1 := #diff, in2 := #minDiff)
      { S7_GenerateENO := "TRUE" } Move(in := #diff, out1 => #minDiff)
      { S7_GenerateENO := "TRUE" } Move(in := 8, out1 => #nextTarget)
   END_RUNG
   // the same network as SCL:
   // ENO of a box is taken as its EN; it also drops when the box reports an error
   IF #req[8] THEN
       #temp1 := 8 - #current;
       #diff := ABS(#temp1);
   END_IF;
   #_w1 := #req[8] AND (#diff < #minDiff);
   IF #_w1 THEN
       #minDiff := #diff;
       #nextTarget := 8;
   END_IF;
END_REGION

REGION Network 11
   RUNG wire#powerrail
      Contact( #req[9] )
      { S7_GenerateENO := "TRUE" } Sub(in1 := 9, in2 := #current, out => #temp1)
      { S7_Templates := "SrcType := Int"; S7_GenerateENO := "TRUE" } Abs(in := #temp1, out => #diff)
      { S7_Templates := "SrcType := Int" } LT_Contact(in1 := #diff, in2 := #minDiff)
      { S7_GenerateENO := "TRUE" } Move(in := #diff, out1 => #minDiff)
      { S7_GenerateENO := "TRUE" } Move(in := 9, out1 => #nextTarget)
   END_RUNG
   // the same network as SCL:
   // ENO of a box is taken as its EN; it also drops when the box reports an error
   IF #req[9] THEN
       #temp1 := 9 - #current;
       #diff := ABS(#temp1);
   END_IF;
   #_w1 := #req[9] AND (#diff < #minDiff);
   IF #_w1 THEN
       #minDiff := #diff;
       #nextTarget := 9;
   END_IF;
END_REGION

REGION Network 12
   RUNG wire#powerrail
      Contact( #req[10] )
      { S7_GenerateENO := "TRUE" } Sub(in1 := 10, in2 := #current, out => #temp1)
      { S7_Templates := "SrcType := Int"; S7_GenerateENO := "TRUE" } Abs(in := #temp1, out => #diff)
      { S7_Templates := "SrcType := Int" } LT_Contact(in1 := #diff, in2 := #minDiff)
      { S7_GenerateENO := "TRUE" } Move(in := #diff, out1 => #minDiff)
      { S7_GenerateENO := "TRUE" } Move(in := 10, out1 => #nextTarget)
   END_RUNG
   // the same network as SCL:
   // ENO of a box is taken as its EN; it also drops when the box reports an error
   IF #req[10] THEN
       #temp1 := 10 - #current;
       #diff := ABS(#temp1);
   END_IF;
   #_w1 := #req[10] AND (#diff < #minDiff);
   IF #_w1 THEN
       #minDiff := #diff;
       #nextTarget := 10;
   END_IF;
END_REGION

REGION Network 13
   RUNG wire#powerrail
      { S7_GenerateENO := "TRUE" } Move(in := #nextTarget, out1 => #GetNextTarget)
   END_RUNG
   // the same network as SCL:
   #GetNextTarget := #nextTarget;
END_REGION
END_FUNCTION

ORGANIZATION_BLOCK "Main"   // OB1, LAD, ProgramCycle
TITLE = "Main Program Sweep (Cycle)"
{ S7_Optimized_Access := 'TRUE' }
VERSION : 0.1
   VAR_TEMP
      RET_VAL : Int;
      RET_VAL_1 : Bool;
      flooradded : Bool;
      floorsubtracted : Bool;
      temp1 : Int;
   END_VAR
   VAR_TEMP   // added for the SCL form of the ladder/FBD networks
      _w1 : Bool;
      _w2 : Bool;
      _w3 : Bool;
      _w4 : Bool;
      _w5 : Bool;
      _w6 : Bool;
   END_VAR
BEGIN

REGION Network 1
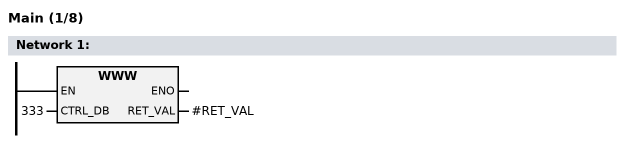
   #RET_VAL := WWW(CTRL_DB := 333);
END_REGION

REGION Network 2
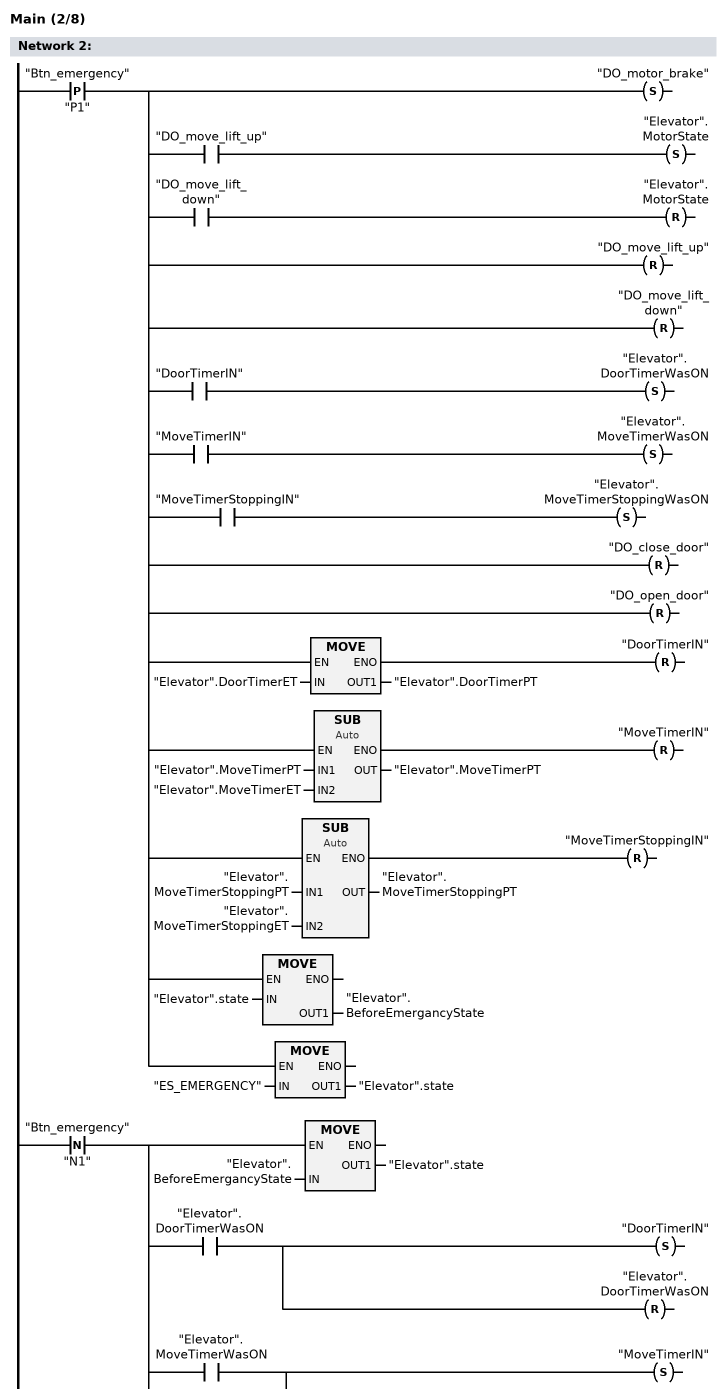
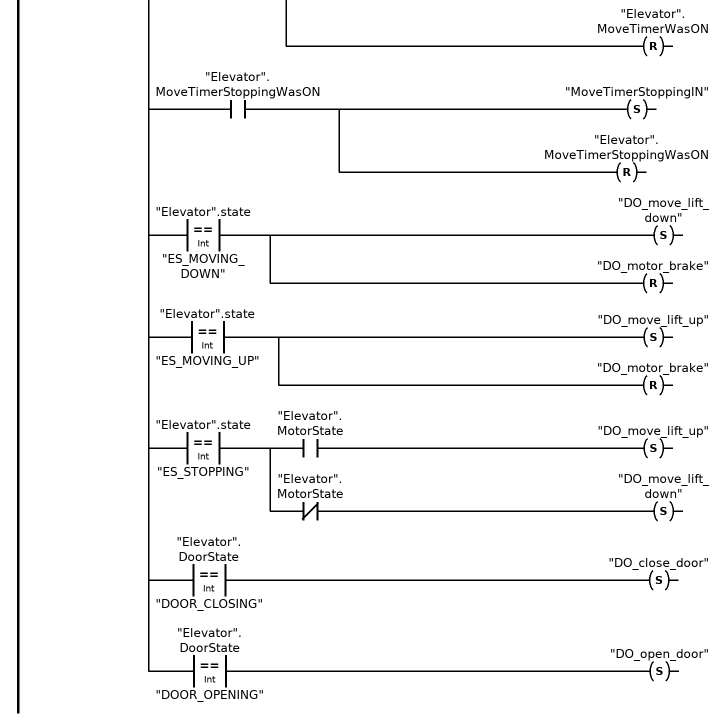
   RUNG wire#powerrail
      P_Contact(operand := "Btn_emergency", bit := "P1")
      wire#w1
      S_Coil( "DO_motor_brake" )
   END_RUNG
   RUNG wire#w1
      Contact( "DO_move_lift_up" )
      S_Coil( "Elevator".MotorState )
   END_RUNG
   RUNG wire#w1
      Contact( "DO_move_lift_down" )
      R_Coil( "Elevator".MotorState )
   END_RUNG
   RUNG wire#w1
      R_Coil( "DO_move_lift_up" )
   END_RUNG
   RUNG wire#w1
      R_Coil( "DO_move_lift_down" )
   END_RUNG
   RUNG wire#w1
      Contact( "DoorTimerIN" )
      S_Coil( "Elevator".DoorTimerWasON )
   END_RUNG
   RUNG wire#w1
      Contact( "MoveTimerIN" )
      S_Coil( "Elevator".MoveTimerWasON )
   END_RUNG
   RUNG wire#w1
      Contact( "MoveTimerStoppingIN" )
      S_Coil( "Elevator".MoveTimerStoppingWasON )
   END_RUNG
   RUNG wire#w1
      R_Coil( "DO_close_door" )
   END_RUNG
   RUNG wire#w1
      R_Coil( "DO_open_door" )
   END_RUNG
   RUNG wire#w1
      Move(in := "Elevator".DoorTimerET, out1 => "Elevator".DoorTimerPT)
      R_Coil( "DoorTimerIN" )
   END_RUNG
   RUNG wire#w1
      Sub(in1 := "Elevator".MoveTimerPT, in2 := "Elevator".MoveTimerET, out => "Elevator".MoveTimerPT)
      R_Coil( "MoveTimerIN" )
   END_RUNG
   RUNG wire#w1
      Sub(in1 := "Elevator".MoveTimerStoppingPT, in2 := "Elevator".MoveTimerStoppingET, out => "Elevator".MoveTimerStoppingPT)
      R_Coil( "MoveTimerStoppingIN" )
   END_RUNG
   RUNG wire#w1
      Move(in := "Elevator".state, out1 => "Elevator".BeforeEmergancyState)
   END_RUNG
   RUNG wire#w1
      Move(in := "ES_EMERGENCY", out1 => "Elevator".state)
   END_RUNG
   RUNG wire#powerrail
      N_Contact(operand := "Btn_emergency", bit := "N1")
      wire#w2
      Move(in := "Elevator".BeforeEmergancyState, out1 => "Elevator".state)
   END_RUNG
   RUNG wire#w2
      Contact( "Elevator".DoorTimerWasON )
      wire#w3
      S_Coil( "DoorTimerIN" )
   END_RUNG
   RUNG wire#w3
      R_Coil( "Elevator".DoorTimerWasON )
   END_RUNG
   RUNG wire#w2
      Contact( "Elevator".MoveTimerWasON )
      wire#w4
      S_Coil( "MoveTimerIN" )
   END_RUNG
   RUNG wire#w4
      R_Coil( "Elevator".MoveTimerWasON )
   END_RUNG
   RUNG wire#w2
      Contact( "Elevator".MoveTimerStoppingWasON )
      wire#w5
      S_Coil( "MoveTimerStoppingIN" )
   END_RUNG
   RUNG wire#w5
      R_Coil( "Elevator".MoveTimerStoppingWasON )
   END_RUNG
   RUNG wire#w2
      { S7_Templates := "SrcType := Int" } EQ_Contact(in1 := "Elevator".state, in2 := "ES_MOVING_DOWN")
      wire#w6
      S_Coil( "DO_move_lift_down" )
   END_RUNG
   RUNG wire#w6
      R_Coil( "DO_motor_brake" )
   END_RUNG
   RUNG wire#w2
      { S7_Templates := "SrcType := Int" } EQ_Contact(in1 := "Elevator".state, in2 := "ES_MOVING_UP")
      wire#w7
      S_Coil( "DO_move_lift_up" )
   END_RUNG
   RUNG wire#w7
      R_Coil( "DO_motor_brake" )
   END_RUNG
   RUNG wire#w2
      { S7_Templates := "SrcType := Int" } EQ_Contact(in1 := "Elevator".state, in2 := "ES_STOPPING")
      wire#w8
      Contact( "Elevator".MotorState )
      S_Coil( "DO_move_lift_up" )
   END_RUNG
   RUNG wire#w8
      I_Contact( "Elevator".MotorState )
      S_Coil( "DO_move_lift_down" )
   END_RUNG
   RUNG wire#w2
      { S7_Templates := "SrcType := Int" } EQ_Contact(in1 := "Elevator".DoorState, in2 := "DOOR_CLOSING")
      S_Coil( "DO_close_door" )
   END_RUNG
   RUNG wire#w2
      { S7_Templates := "SrcType := Int" } EQ_Contact(in1 := "Elevator".DoorState, in2 := "DOOR_OPENING")
      S_Coil( "DO_open_door" )
   END_RUNG
   // the same network as SCL:
   #_w1 := "Btn_emergency" AND NOT "P1";   // rising edge of "Btn_emergency"
   "P1" := "Btn_emergency";
   IF #_w1 THEN "DO_motor_brake" := TRUE; END_IF;
   IF #_w1 AND "DO_move_lift_up" THEN "Elevator".MotorState := TRUE; END_IF;
   IF #_w1 AND "DO_move_lift_down" THEN "Elevator".MotorState := FALSE; END_IF;
   IF #_w1 THEN
       "DO_move_lift_up" := FALSE;
       "DO_move_lift_down" := FALSE;
   END_IF;
   IF #_w1 AND "DoorTimerIN" THEN "Elevator".DoorTimerWasON := TRUE; END_IF;
   IF #_w1 AND "MoveTimerIN" THEN "Elevator".MoveTimerWasON := TRUE; END_IF;
   IF #_w1 AND "MoveTimerStoppingIN" THEN "Elevator".MoveTimerStoppingWasON := TRUE; END_IF;
   IF #_w1 THEN
       "DO_close_door" := FALSE;
       "DO_open_door" := FALSE;
       "Elevator".DoorTimerPT := "Elevator".DoorTimerET;
       "DoorTimerIN" := FALSE;
       "Elevator".MoveTimerPT := "Elevator".MoveTimerPT - "Elevator".MoveTimerET;
       "MoveTimerIN" := FALSE;
       "Elevator".MoveTimerStoppingPT := "Elevator".MoveTimerStoppingPT - "Elevator".MoveTimerStoppingET;
       "MoveTimerStoppingIN" := FALSE;
       "Elevator".BeforeEmergancyState := "Elevator".state;
       "Elevator".state := "ES_EMERGENCY";
   END_IF;
   #_w2 := NOT "Btn_emergency" AND "N1";   // falling edge of "Btn_emergency"
   "N1" := "Btn_emergency";
   IF #_w2 THEN "Elevator".state := "Elevator".BeforeEmergancyState; END_IF;
   IF #_w2 AND "Elevator".DoorTimerWasON THEN
       "DoorTimerIN" := TRUE;
       "Elevator".DoorTimerWasON := FALSE;
   END_IF;
   IF #_w2 AND "Elevator".MoveTimerWasON THEN
       "MoveTimerIN" := TRUE;
       "Elevator".MoveTimerWasON := FALSE;
   END_IF;
   IF #_w2 AND "Elevator".MoveTimerStoppingWasON THEN
       "MoveTimerStoppingIN" := TRUE;
       "Elevator".MoveTimerStoppingWasON := FALSE;
   END_IF;
   IF #_w2 AND ("Elevator".state = "ES_MOVING_DOWN") THEN
       "DO_move_lift_down" := TRUE;
       "DO_motor_brake" := FALSE;
   END_IF;
   IF #_w2 AND ("Elevator".state = "ES_MOVING_UP") THEN
       "DO_move_lift_up" := TRUE;
       "DO_motor_brake" := FALSE;
   END_IF;
   #_w3 := #_w2 AND ("Elevator".state = "ES_STOPPING");
   IF #_w3 AND "Elevator".MotorState THEN "DO_move_lift_up" := TRUE; END_IF;
   IF #_w3 AND NOT "Elevator".MotorState THEN "DO_move_lift_down" := TRUE; END_IF;
   IF #_w2 AND ("Elevator".DoorState = "DOOR_CLOSING") THEN "DO_close_door" := TRUE; END_IF;
   IF #_w2 AND ("Elevator".DoorState = "DOOR_OPENING") THEN "DO_open_door" := TRUE; END_IF;
END_REGION

REGION Network 3
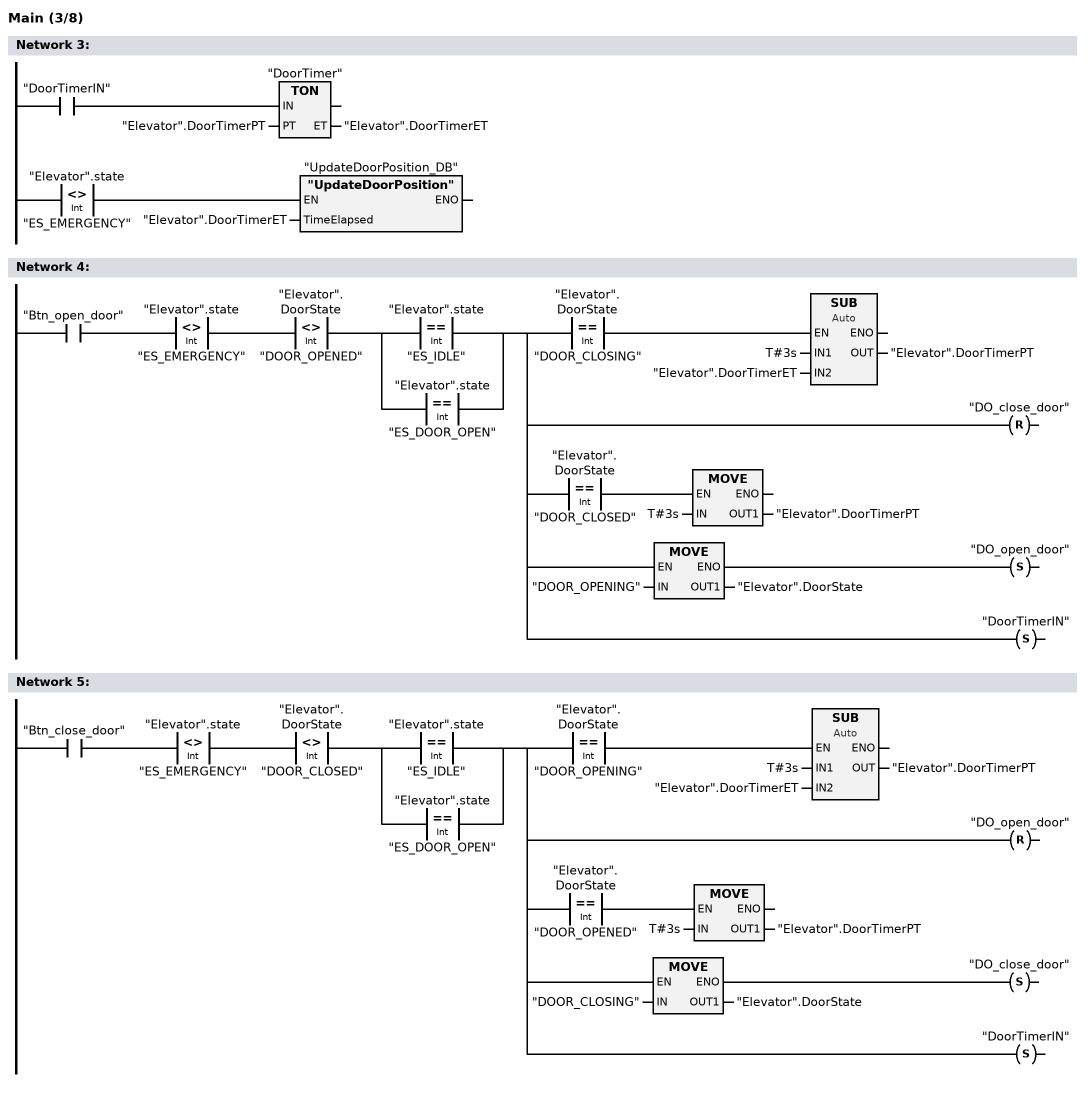
   "DoorTimer".TON(IN := "DoorTimerIN", PT := "Elevator".DoorTimerPT, ET => "Elevator".DoorTimerET);
   IF "Elevator".state <> "ES_EMERGENCY" THEN
       "UpdateDoorPosition_DB"(TimeElapsed := "Elevator".DoorTimerET);   // "UpdateDoorPosition"
   END_IF;
END_REGION

REGION Network 4
   RUNG wire#powerrail
      Contact( "Btn_open_door" )
      { S7_Templates := "SrcType := Int" } NE_Contact(in1 := "Elevator".state, in2 := "ES_EMERGENCY")
      { S7_Templates := "SrcType := Int" } NE_Contact(in1 := "Elevator".DoorState, in2 := "DOOR_OPENED")
      wire#w1
      { S7_Templates := "SrcType := Int" } EQ_Contact(in1 := "Elevator".state, in2 := "ES_IDLE")
      wire#w2
      { S7_Templates := "SrcType := Int" } EQ_Contact(in1 := "Elevator".DoorState, in2 := "DOOR_CLOSING")
      Sub(in1 := T#3s, in2 := "Elevator".DoorTimerET, out => "Elevator".DoorTimerPT)
   END_RUNG
   RUNG wire#w1
      { S7_Templates := "SrcType := Int" } EQ_Contact(in1 := "Elevator".state, in2 := "ES_DOOR_OPEN")
   END_RUNG wire#w2
   RUNG wire#w2
      R_Coil( "DO_close_door" )
   END_RUNG
   RUNG wire#w2
      { S7_Templates := "SrcType := Int" } EQ_Contact(in1 := "Elevator".DoorState, in2 := "DOOR_CLOSED")
      Move(in := T#3s, out1 => "Elevator".DoorTimerPT)
   END_RUNG
   RUNG wire#w2
      Move(in := "DOOR_OPENING", out1 => "Elevator".DoorState)
      S_Coil( "DO_open_door" )
   END_RUNG
   RUNG wire#w2
      S_Coil( "DoorTimerIN" )
   END_RUNG
   // the same network as SCL:
   #_w1 := "Btn_open_door" AND ("Elevator".state <> "ES_EMERGENCY") AND ("Elevator".DoorState <> "DOOR_OPENED") AND (("Elevator".state = "ES_IDLE") OR ("Elevator".state = "ES_DOOR_OPEN"));
   IF #_w1 AND ("Elevator".DoorState = "DOOR_CLOSING") THEN
       "Elevator".DoorTimerPT := T#3s - "Elevator".DoorTimerET;
   END_IF;
   IF #_w1 THEN "DO_close_door" := FALSE; END_IF;
   IF #_w1 AND ("Elevator".DoorState = "DOOR_CLOSED") THEN "Elevator".DoorTimerPT := T#3s; END_IF;
   IF #_w1 THEN
       "Elevator".DoorState := "DOOR_OPENING";
       "DO_open_door" := TRUE;
       "DoorTimerIN" := TRUE;
   END_IF;
END_REGION

REGION Network 5
   RUNG wire#powerrail
      Contact( "Btn_close_door" )
      { S7_Templates := "SrcType := Int" } NE_Contact(in1 := "Elevator".state, in2 := "ES_EMERGENCY")
      { S7_Templates := "SrcType := Int" } NE_Contact(in1 := "Elevator".DoorState, in2 := "DOOR_CLOSED")
      wire#w1
      { S7_Templates := "SrcType := Int" } EQ_Contact(in1 := "Elevator".state, in2 := "ES_IDLE")
      wire#w2
      { S7_Templates := "SrcType := Int" } EQ_Contact(in1 := "Elevator".DoorState, in2 := "DOOR_OPENING")
      Sub(in1 := T#3s, in2 := "Elevator".DoorTimerET, out => "Elevator".DoorTimerPT)
   END_RUNG
   RUNG wire#w1
      { S7_Templates := "SrcType := Int" } EQ_Contact(in1 := "Elevator".state, in2 := "ES_DOOR_OPEN")
   END_RUNG wire#w2
   RUNG wire#w2
      R_Coil( "DO_open_door" )
   END_RUNG
   RUNG wire#w2
      { S7_Templates := "SrcType := Int" } EQ_Contact(in1 := "Elevator".DoorState, in2 := "DOOR_OPENED")
      Move(in := T#3s, out1 => "Elevator".DoorTimerPT)
   END_RUNG
   RUNG wire#w2
      Move(in := "DOOR_CLOSING", out1 => "Elevator".DoorState)
      S_Coil( "DO_close_door" )
   END_RUNG
   RUNG wire#w2
      S_Coil( "DoorTimerIN" )
   END_RUNG
   // the same network as SCL:
   #_w1 := "Btn_close_door" AND ("Elevator".state <> "ES_EMERGENCY") AND ("Elevator".DoorState <> "DOOR_CLOSED") AND (("Elevator".state = "ES_IDLE") OR ("Elevator".state = "ES_DOOR_OPEN"));
   IF #_w1 AND ("Elevator".DoorState = "DOOR_OPENING") THEN
       "Elevator".DoorTimerPT := T#3s - "Elevator".DoorTimerET;
   END_IF;
   IF #_w1 THEN "DO_open_door" := FALSE; END_IF;
   IF #_w1 AND ("Elevator".DoorState = "DOOR_OPENED") THEN "Elevator".DoorTimerPT := T#3s; END_IF;
   IF #_w1 THEN
       "Elevator".DoorState := "DOOR_CLOSING";
       "DO_close_door" := TRUE;
       "DoorTimerIN" := TRUE;
   END_IF;
END_REGION

REGION Network 6
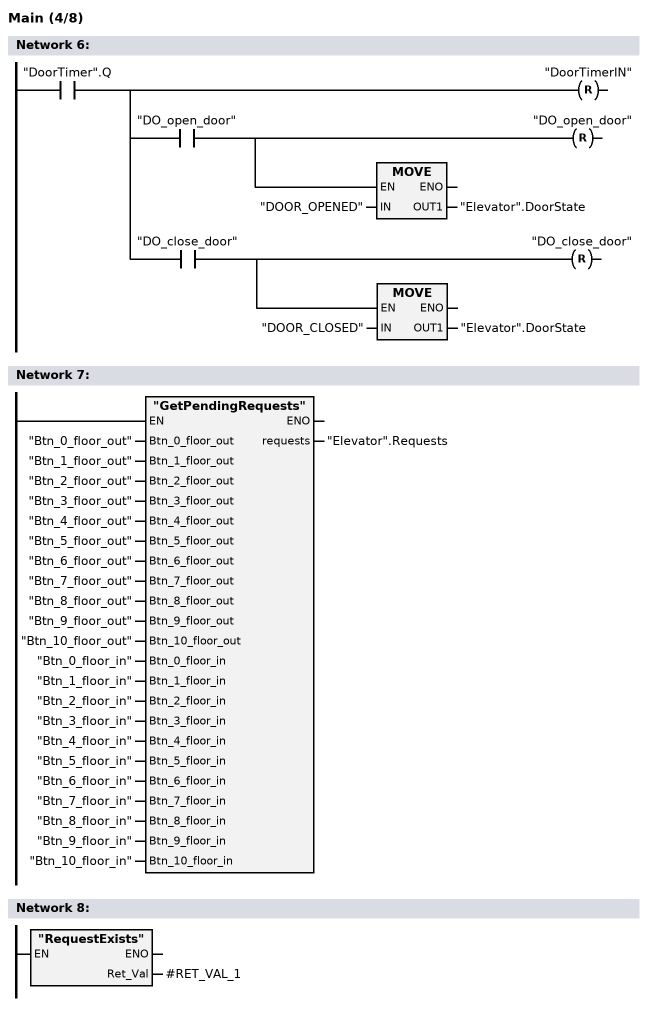
   RUNG wire#powerrail
      Contact( "DoorTimer".Q )
      wire#w1
      R_Coil( "DoorTimerIN" )
   END_RUNG
   RUNG wire#w1
      Contact( "DO_open_door" )
      wire#w2
      R_Coil( "DO_open_door" )
   END_RUNG
   RUNG wire#w2
      Move(in := "DOOR_OPENED", out1 => "Elevator".DoorState)
   END_RUNG
   RUNG wire#w1
      Contact( "DO_close_door" )
      wire#w3
      R_Coil( "DO_close_door" )
   END_RUNG
   RUNG wire#w3
      Move(in := "DOOR_CLOSED", out1 => "Elevator".DoorState)
   END_RUNG
   // the same network as SCL:
   IF "DoorTimer".Q THEN "DoorTimerIN" := FALSE; END_IF;
   #_w1 := "DoorTimer".Q AND "DO_open_door";
   IF #_w1 THEN
       "DO_open_door" := FALSE;
       "Elevator".DoorState := "DOOR_OPENED";
   END_IF;
   #_w2 := "DoorTimer".Q AND "DO_close_door";
   IF #_w2 THEN
       "DO_close_door" := FALSE;
       "Elevator".DoorState := "DOOR_CLOSED";
   END_IF;
END_REGION

REGION Network 7
   RUNG wire#powerrail
      "GetPendingRequests"(Btn_0_floor_out := "Btn_0_floor_out", Btn_1_floor_out := "Btn_1_floor_out", Btn_2_floor_out := "Btn_2_floor_out", Btn_3_floor_out := "Btn_3_floor_out", Btn_4_floor_out := "Btn_4_floor_out", Btn_5_floor_out := "Btn_5_floor_out", Btn_6_floor_out := "Btn_6_floor_out", Btn_7_floor_out := "Btn_7_floor_out", Btn_8_floor_out := "Btn_8_floor_out", Btn_9_floor_out := "Btn_9_floor_out", Btn_10_floor_out := "Btn_10_floor_out", Btn_0_floor_in := "Btn_0_floor_in", Btn_1_floor_in := "Btn_1_floor_in", Btn_2_floor_in := "Btn_2_floor_in", Btn_3_floor_in := "Btn_3_floor_in", Btn_4_floor_in := "Btn_4_floor_in", Btn_5_floor_in := "Btn_5_floor_in", Btn_6_floor_in := "Btn_6_floor_in", Btn_7_floor_in := "Btn_7_floor_in", Btn_8_floor_in := "Btn_8_floor_in", Btn_9_floor_in := "Btn_9_floor_in", Btn_10_floor_in := "Btn_10_floor_in", requests => "Elevator".Requests)
   END_RUNG
   // the same network as SCL:
   "GetPendingRequests"(Btn_0_floor_out := "Btn_0_floor_out",
                        Btn_1_floor_out := "Btn_1_floor_out",
                        Btn_2_floor_out := "Btn_2_floor_out",
                        Btn_3_floor_out := "Btn_3_floor_out",
                        Btn_4_floor_out := "Btn_4_floor_out",
                        Btn_5_floor_out := "Btn_5_floor_out",
                        Btn_6_floor_out := "Btn_6_floor_out",
                        Btn_7_floor_out := "Btn_7_floor_out",
                        Btn_8_floor_out := "Btn_8_floor_out",
                        Btn_9_floor_out := "Btn_9_floor_out",
                        Btn_10_floor_out := "Btn_10_floor_out",
                        Btn_0_floor_in := "Btn_0_floor_in",
                        Btn_1_floor_in := "Btn_1_floor_in",
                        Btn_2_floor_in := "Btn_2_floor_in",
                        Btn_3_floor_in := "Btn_3_floor_in",
                        Btn_4_floor_in := "Btn_4_floor_in",
                        Btn_5_floor_in := "Btn_5_floor_in",
                        Btn_6_floor_in := "Btn_6_floor_in",
                        Btn_7_floor_in := "Btn_7_floor_in",
                        Btn_8_floor_in := "Btn_8_floor_in",
                        Btn_9_floor_in := "Btn_9_floor_in",
                        Btn_10_floor_in := "Btn_10_floor_in",
                        requests => "Elevator".Requests);
END_REGION

REGION Network 8
   RUNG wire#powerrail
      "RequestExists"(Ret_Val => #RET_VAL_1)
   END_RUNG
   // the same network as SCL:
   #RET_VAL_1 := "RequestExists"();
END_REGION

REGION Network 9
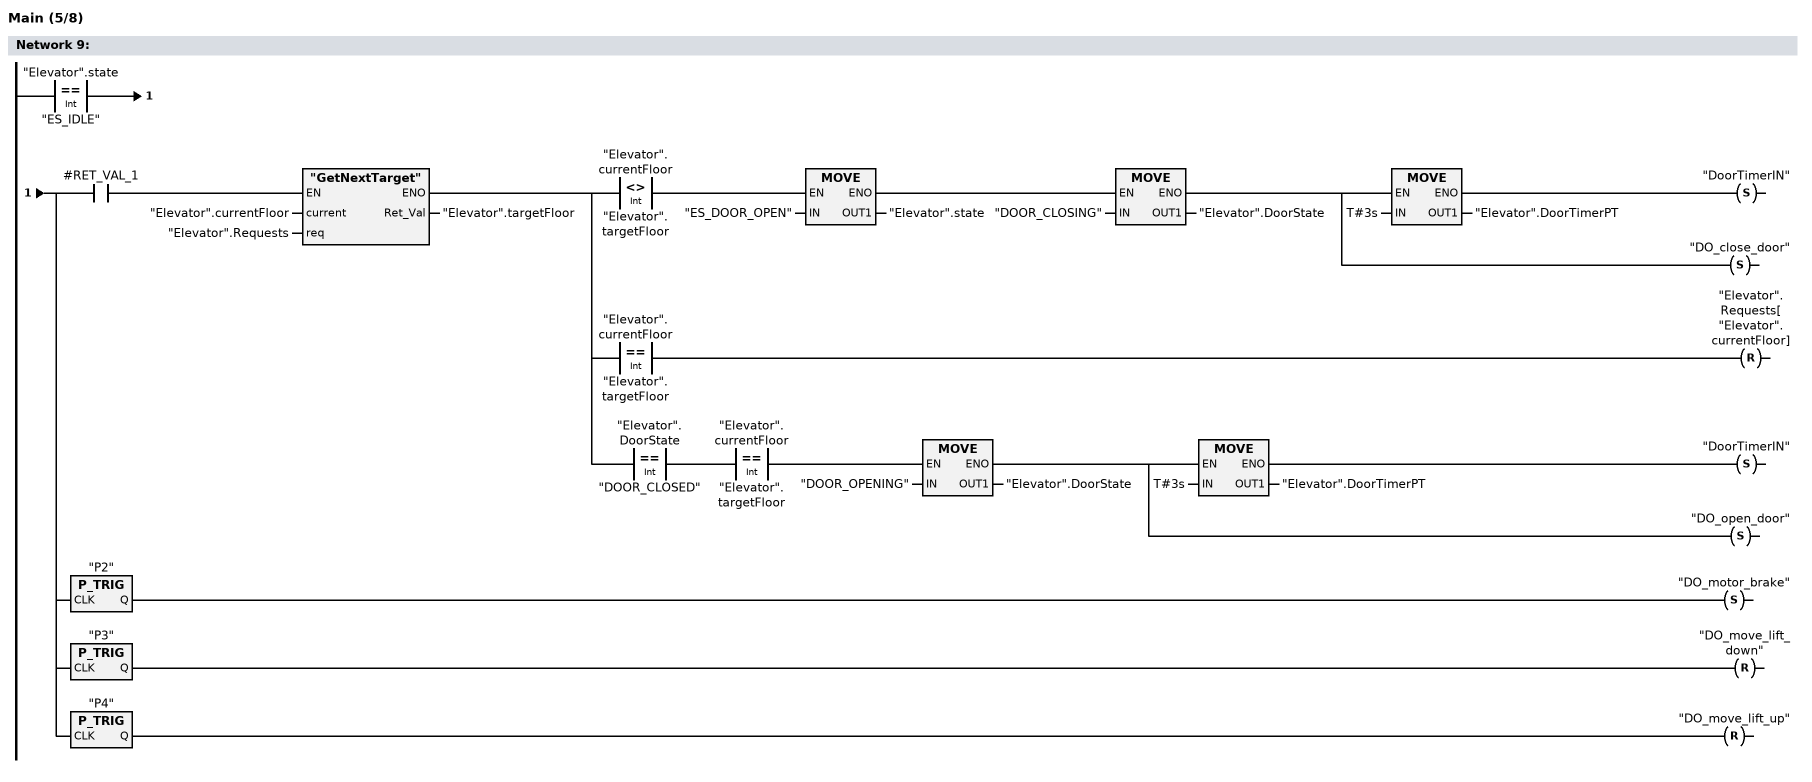
   RUNG wire#powerrail
      { S7_Templates := "SrcType := Int" } EQ_Contact(in1 := "Elevator".state, in2 := "ES_IDLE")
      wire#w1
      Contact( #RET_VAL_1 )
      "GetNextTarget"(current := "Elevator".currentFloor, req := "Elevator".Requests, Ret_Val => "Elevator".targetFloor)
      wire#w2
      { S7_Templates := "SrcType := Int" } NE_Contact(in1 := "Elevator".currentFloor, in2 := "Elevator".targetFloor)
      { S7_GenerateENO := "TRUE" } Move(in := "ES_DOOR_OPEN", out1 => "Elevator".state)
      { S7_GenerateENO := "TRUE" } Move(in := "DOOR_CLOSING", out1 => "Elevator".DoorState)
      wire#w3
      { S7_GenerateENO := "TRUE" } Move(in := T#3s, out1 => "Elevator".DoorTimerPT)
      S_Coil( "DoorTimerIN" )
   END_RUNG
   RUNG wire#w3
      S_Coil( "DO_close_door" )
   END_RUNG
   RUNG wire#w2
      { S7_Templates := "SrcType := Int" } EQ_Contact(in1 := "Elevator".currentFloor, in2 := "Elevator".targetFloor)
      R_Coil( "Elevator".Requests["Elevator".currentFloor] )
   END_RUNG
   RUNG wire#w2
      { S7_Templates := "SrcType := Int" } EQ_Contact(in1 := "Elevator".DoorState, in2 := "DOOR_CLOSED")
      { S7_Templates := "SrcType := Int" } EQ_Contact(in1 := "Elevator".currentFloor, in2 := "Elevator".targetFloor)
      { S7_GenerateENO := "TRUE" } Move(in := "DOOR_OPENING", out1 => "Elevator".DoorState)
      wire#w4
      { S7_GenerateENO := "TRUE" } Move(in := T#3s, out1 => "Elevator".DoorTimerPT)
      S_Coil( "DoorTimerIN" )
   END_RUNG
   RUNG wire#w4
      S_Coil( "DO_open_door" )
   END_RUNG
   RUNG wire#w1
      P_Trig( "P2" )
      S_Coil( "DO_motor_brake" )
   END_RUNG
   RUNG wire#w1
      P_Trig( "P3" )
      R_Coil( "DO_move_lift_down" )
   END_RUNG
   RUNG wire#w1
      P_Trig( "P4" )
      R_Coil( "DO_move_lift_up" )
   END_RUNG
   // the same network as SCL:
   // ENO of a box is taken as its EN; it also drops when the box reports an error
   #_w1 := "Elevator".state = "ES_IDLE";
   "Elevator".targetFloor := "GetNextTarget"(EN := #_w1 AND #RET_VAL_1,
                           current := "Elevator".currentFloor,
                           req := "Elevator".Requests,
                           ENO => #_w2);
   IF #_w2 AND ("Elevator".currentFloor <> "Elevator".targetFloor) THEN
       "Elevator".state := "ES_DOOR_OPEN";
       "Elevator".DoorState := "DOOR_CLOSING";
       "Elevator".DoorTimerPT := T#3s;
       "DoorTimerIN" := TRUE;
       "DO_close_door" := TRUE;
   END_IF;
   IF #_w2 AND ("Elevator".currentFloor = "Elevator".targetFloor) THEN
       "Elevator".Requests["Elevator".currentFloor] := FALSE;
   END_IF;
   #_w3 := #_w2 AND ("Elevator".DoorState = "DOOR_CLOSED") AND ("Elevator".currentFloor = "Elevator".targetFloor);
   IF #_w3 THEN
       "Elevator".DoorState := "DOOR_OPENING";
       "Elevator".DoorTimerPT := T#3s;
       "DoorTimerIN" := TRUE;
       "DO_open_door" := TRUE;
   END_IF;
   #_w4 := #_w1 AND NOT "P2";   // rising edge
   "P2" := #_w1;
   IF #_w4 THEN "DO_motor_brake" := TRUE; END_IF;
   #_w5 := #_w1 AND NOT "P3";   // rising edge
   "P3" := #_w1;
   IF #_w5 THEN "DO_move_lift_down" := FALSE; END_IF;
   #_w6 := #_w1 AND NOT "P4";   // rising edge
   "P4" := #_w1;
   IF #_w6 THEN "DO_move_lift_up" := FALSE; END_IF;
END_REGION

REGION Network 10
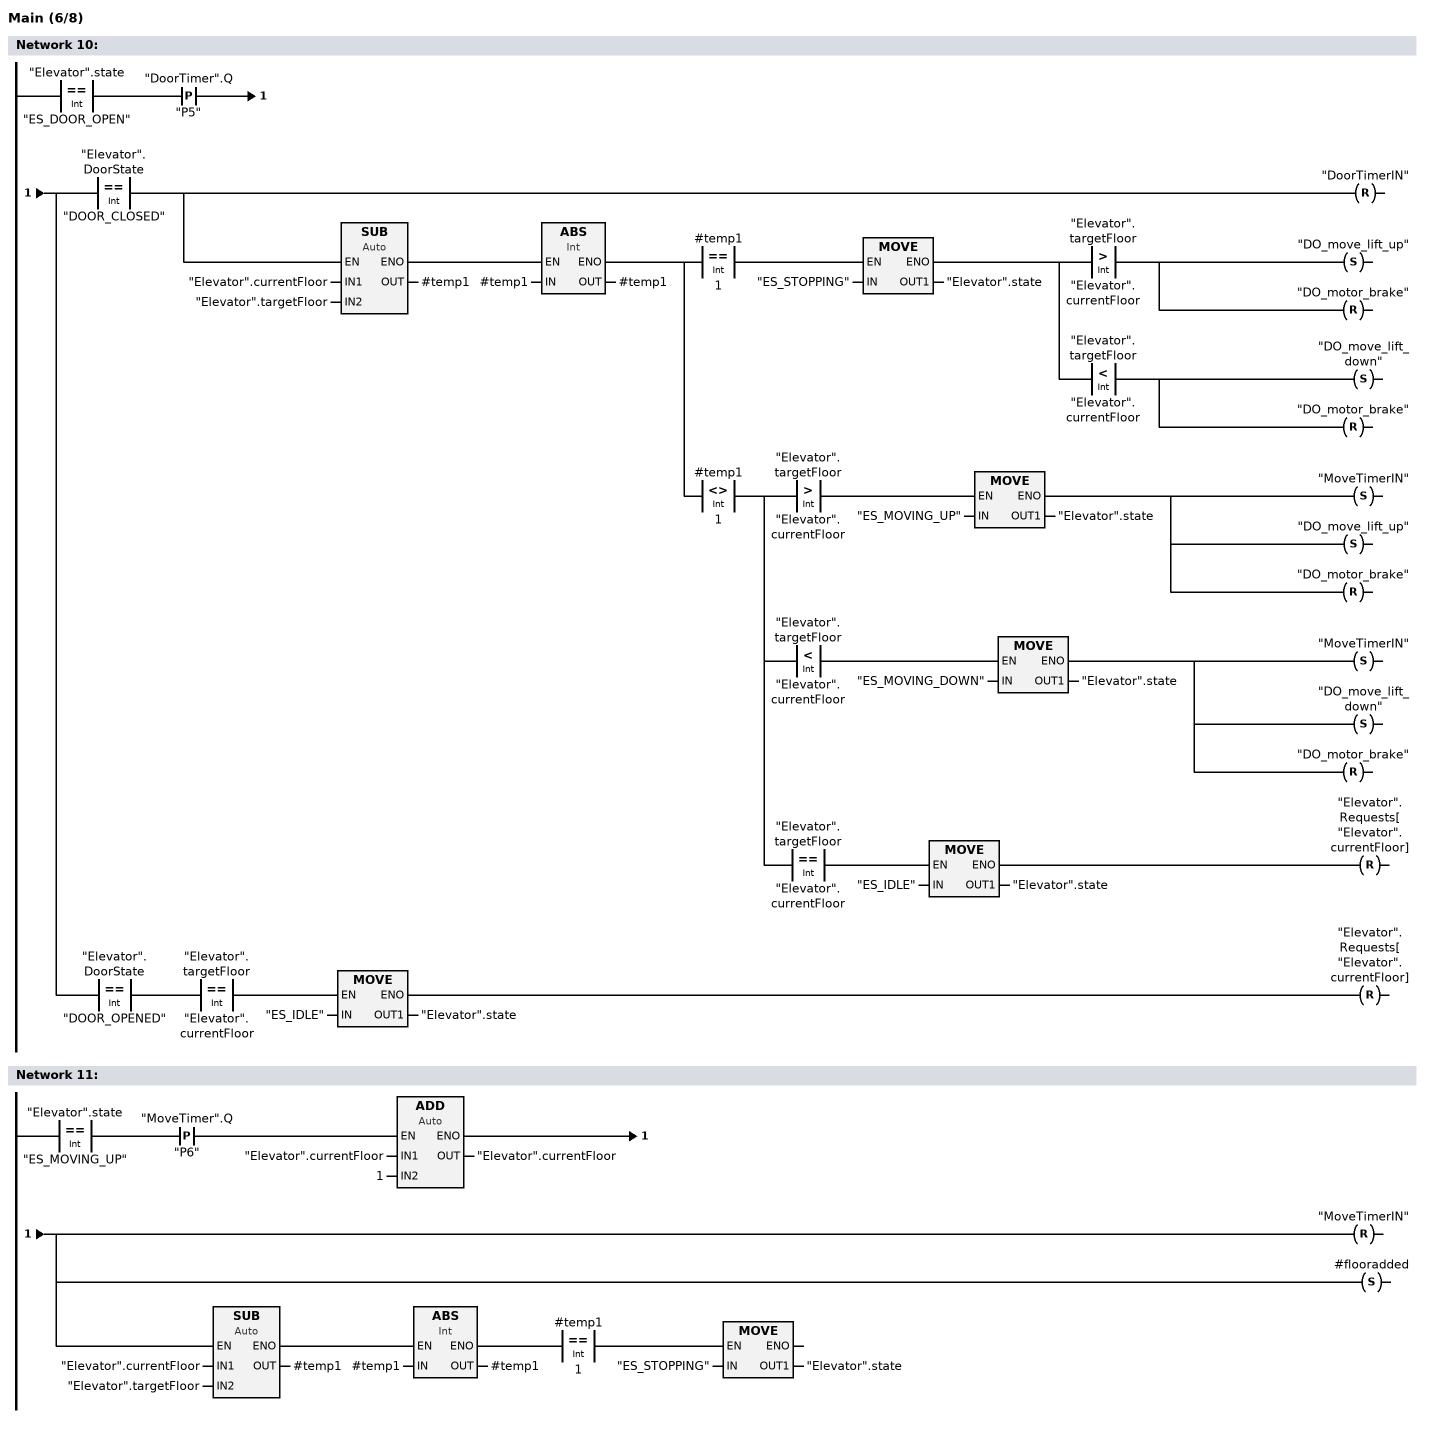
   RUNG wire#powerrail
      { S7_Templates := "SrcType := Int" } EQ_Contact(in1 := "Elevator".state, in2 := "ES_DOOR_OPEN")
      P_Contact(operand := "DoorTimer".Q, bit := "P5")
      wire#w1
      { S7_Templates := "SrcType := Int" } EQ_Contact(in1 := "Elevator".DoorState, in2 := "DOOR_CLOSED")
      wire#w2
      R_Coil( "DoorTimerIN" )
   END_RUNG
   RUNG wire#w2
      Sub(in1 := "Elevator".currentFloor, in2 := "Elevator".targetFloor, out => #temp1)
      { S7_Templates := "SrcType := Int" } Abs(in := #temp1, out => #temp1)
      wire#w3
      { S7_Templates := "SrcType := Int" } EQ_Contact(in1 := #temp1, in2 := 1)
      { S7_GenerateENO := "TRUE" } Move(in := "ES_STOPPING", out1 => "Elevator".state)
      wire#w4
      { S7_Templates := "SrcType := Int" } GT_Contact(in1 := "Elevator".targetFloor, in2 := "Elevator".currentFloor)
      wire#w5
      S_Coil( "DO_move_lift_up" )
   END_RUNG
   RUNG wire#w5
      R_Coil( "DO_motor_brake" )
   END_RUNG
   RUNG wire#w4
      { S7_Templates := "SrcType := Int" } LT_Contact(in1 := "Elevator".targetFloor, in2 := "Elevator".currentFloor)
      wire#w6
      S_Coil( "DO_move_lift_down" )
   END_RUNG
   RUNG wire#w6
      R_Coil( "DO_motor_brake" )
   END_RUNG
   RUNG wire#w3
      { S7_Templates := "SrcType := Int" } NE_Contact(in1 := #temp1, in2 := 1)
      wire#w7
      { S7_Templates := "SrcType := Int" } GT_Contact(in1 := "Elevator".targetFloor, in2 := "Elevator".currentFloor)
      { S7_GenerateENO := "TRUE" } Move(in := "ES_MOVING_UP", out1 => "Elevator".state)
      wire#w8
      S_Coil( "MoveTimerIN" )
   END_RUNG
   RUNG wire#w8
      S_Coil( "DO_move_lift_up" )
   END_RUNG
   RUNG wire#w8
      R_Coil( "DO_motor_brake" )
   END_RUNG
   RUNG wire#w7
      { S7_Templates := "SrcType := Int" } LT_Contact(in1 := "Elevator".targetFloor, in2 := "Elevator".currentFloor)
      { S7_GenerateENO := "TRUE" } Move(in := "ES_MOVING_DOWN", out1 => "Elevator".state)
      wire#w9
      S_Coil( "MoveTimerIN" )
   END_RUNG
   RUNG wire#w9
      S_Coil( "DO_move_lift_down" )
   END_RUNG
   RUNG wire#w9
      R_Coil( "DO_motor_brake" )
   END_RUNG
   RUNG wire#w7
      { S7_Templates := "SrcType := Int" } EQ_Contact(in1 := "Elevator".targetFloor, in2 := "Elevator".currentFloor)
      { S7_GenerateENO := "TRUE" } Move(in := "ES_IDLE", out1 => "Elevator".state)
      R_Coil( "Elevator".Requests["Elevator".currentFloor] )
   END_RUNG
   RUNG wire#w1
      { S7_Templates := "SrcType := Int" } EQ_Contact(in1 := "Elevator".DoorState, in2 := "DOOR_OPENED")
      { S7_Templates := "SrcType := Int" } EQ_Contact(in1 := "Elevator".targetFloor, in2 := "Elevator".currentFloor)
      { S7_GenerateENO := "TRUE" } Move(in := "ES_IDLE", out1 => "Elevator".state)
      R_Coil( "Elevator".Requests["Elevator".currentFloor] )
   END_RUNG
   // the same network as SCL:
   // ENO of a box is taken as its EN; it also drops when the box reports an error
   #_w1 := ("Elevator".state = "ES_DOOR_OPEN") AND "DoorTimer".Q AND NOT "P5";   // rising edge of "DoorTimer".Q
   "P5" := "DoorTimer".Q;
   #_w2 := #_w1 AND ("Elevator".DoorState = "DOOR_CLOSED");
   IF #_w2 THEN
       "DoorTimerIN" := FALSE;
       #temp1 := "Elevator".currentFloor - "Elevator".targetFloor;
       #temp1 := ABS(#temp1);
   END_IF;
   #_w3 := #_w2 AND (#temp1 = 1);
   IF #_w3 THEN "Elevator".state := "ES_STOPPING"; END_IF;
   IF #_w3 AND ("Elevator".targetFloor > "Elevator".currentFloor) THEN
       "DO_move_lift_up" := TRUE;
       "DO_motor_brake" := FALSE;
   END_IF;
   IF #_w3 AND ("Elevator".targetFloor < "Elevator".currentFloor) THEN
       "DO_move_lift_down" := TRUE;
       "DO_motor_brake" := FALSE;
   END_IF;
   #_w4 := #_w2 AND (#temp1 <> 1);
   IF #_w4 AND ("Elevator".targetFloor > "Elevator".currentFloor) THEN
       "Elevator".state := "ES_MOVING_UP";
       "MoveTimerIN" := TRUE;
       "DO_move_lift_up" := TRUE;
       "DO_motor_brake" := FALSE;
   END_IF;
   IF #_w4 AND ("Elevator".targetFloor < "Elevator".currentFloor) THEN
       "Elevator".state := "ES_MOVING_DOWN";
       "MoveTimerIN" := TRUE;
       "DO_move_lift_down" := TRUE;
       "DO_motor_brake" := FALSE;
   END_IF;
   IF #_w4 AND ("Elevator".targetFloor = "Elevator".currentFloor) THEN
       "Elevator".state := "ES_IDLE";
       "Elevator".Requests["Elevator".currentFloor] := FALSE;
   END_IF;
   IF #_w1 AND ("Elevator".DoorState = "DOOR_OPENED") AND ("Elevator".targetFloor = "Elevator".currentFloor) THEN
       "Elevator".state := "ES_IDLE";
       "Elevator".Requests["Elevator".currentFloor] := FALSE;
   END_IF;
END_REGION

REGION Network 11
   RUNG wire#powerrail
      { S7_Templates := "SrcType := Int" } EQ_Contact(in1 := "Elevator".state, in2 := "ES_MOVING_UP")
      P_Contact(operand := "MoveTimer".Q, bit := "P6")
      { S7_GenerateENO := "TRUE" } Add(in1 := "Elevator".currentFloor, in2 := 1, out => "Elevator".currentFloor)
      wire#w1
      R_Coil( "MoveTimerIN" )
   END_RUNG
   RUNG wire#w1
      S_Coil( #flooradded )
   END_RUNG
   RUNG wire#w1
      Sub(in1 := "Elevator".currentFloor, in2 := "Elevator".targetFloor, out => #temp1)
      { S7_Templates := "SrcType := Int" } Abs(in := #temp1, out => #temp1)
      { S7_Templates := "SrcType := Int" } EQ_Contact(in1 := #temp1, in2 := 1)
      { S7_GenerateENO := "TRUE" } Move(in := "ES_STOPPING", out1 => "Elevator".state)
   END_RUNG
   // the same network as SCL:
   // ENO of a box is taken as its EN; it also drops when the box reports an error
   #_w1 := ("Elevator".state = "ES_MOVING_UP") AND "MoveTimer".Q AND NOT "P6";   // rising edge of "MoveTimer".Q
   "P6" := "MoveTimer".Q;
   IF #_w1 THEN
       "Elevator".currentFloor := "Elevator".currentFloor + 1;
       "MoveTimerIN" := FALSE;
       #flooradded := TRUE;
       #temp1 := "Elevator".currentFloor - "Elevator".targetFloor;
       #temp1 := ABS(#temp1);
   END_IF;
   IF #_w1 AND (#temp1 = 1) THEN "Elevator".state := "ES_STOPPING"; END_IF;
END_REGION

REGION Network 12
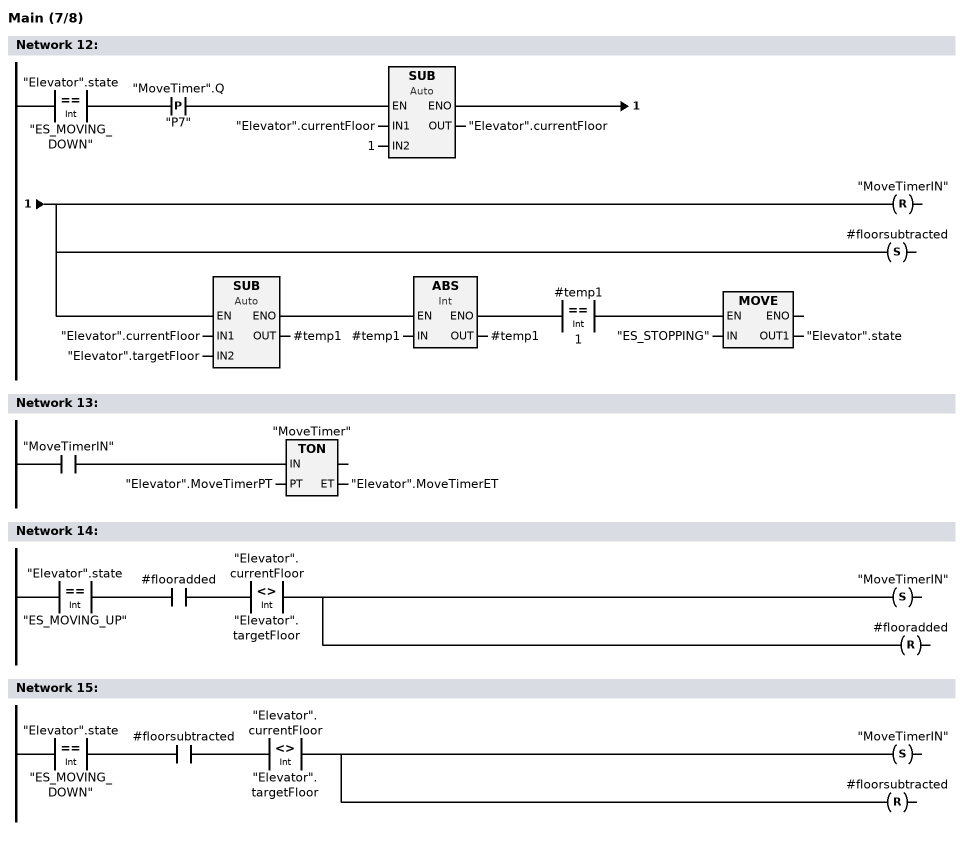
   RUNG wire#powerrail
      { S7_Templates := "SrcType := Int" } EQ_Contact(in1 := "Elevator".state, in2 := "ES_MOVING_DOWN")
      P_Contact(operand := "MoveTimer".Q, bit := "P7")
      { S7_GenerateENO := "TRUE" } Sub(in1 := "Elevator".currentFloor, in2 := 1, out => "Elevator".currentFloor)
      wire#w1
      R_Coil( "MoveTimerIN" )
   END_RUNG
   RUNG wire#w1
      S_Coil( #floorsubtracted )
   END_RUNG
   RUNG wire#w1
      Sub(in1 := "Elevator".currentFloor, in2 := "Elevator".targetFloor, out => #temp1)
      { S7_Templates := "SrcType := Int" } Abs(in := #temp1, out => #temp1)
      { S7_Templates := "SrcType := Int" } EQ_Contact(in1 := #temp1, in2 := 1)
      { S7_GenerateENO := "TRUE" } Move(in := "ES_STOPPING", out1 => "Elevator".state)
   END_RUNG
   // the same network as SCL:
   // ENO of a box is taken as its EN; it also drops when the box reports an error
   #_w1 := ("Elevator".state = "ES_MOVING_DOWN") AND "MoveTimer".Q AND NOT "P7";   // rising edge of "MoveTimer".Q
   "P7" := "MoveTimer".Q;
   IF #_w1 THEN
       "Elevator".currentFloor := "Elevator".currentFloor - 1;
       "MoveTimerIN" := FALSE;
       #floorsubtracted := TRUE;
       #temp1 := "Elevator".currentFloor - "Elevator".targetFloor;
       #temp1 := ABS(#temp1);
   END_IF;
   IF #_w1 AND (#temp1 = 1) THEN "Elevator".state := "ES_STOPPING"; END_IF;
END_REGION

REGION Network 13
   "MoveTimer".TON(IN := "MoveTimerIN", PT := "Elevator".MoveTimerPT, ET => "Elevator".MoveTimerET);
END_REGION

REGION Network 14
   RUNG wire#powerrail
      { S7_Templates := "SrcType := Int" } EQ_Contact(in1 := "Elevator".state, in2 := "ES_MOVING_UP")
      Contact( #flooradded )
      { S7_Templates := "SrcType := Int" } NE_Contact(in1 := "Elevator".currentFloor, in2 := "Elevator".targetFloor)
      wire#w1
      S_Coil( "MoveTimerIN" )
   END_RUNG
   RUNG wire#w1
      R_Coil( #flooradded )
   END_RUNG
   // the same network as SCL:
   IF ("Elevator".state = "ES_MOVING_UP") AND #flooradded AND ("Elevator".currentFloor <> "Elevator".targetFloor) THEN
       "MoveTimerIN" := TRUE;
       #flooradded := FALSE;
   END_IF;
END_REGION

REGION Network 15
   RUNG wire#powerrail
      { S7_Templates := "SrcType := Int" } EQ_Contact(in1 := "Elevator".state, in2 := "ES_MOVING_DOWN")
      Contact( #floorsubtracted )
      { S7_Templates := "SrcType := Int" } NE_Contact(in1 := "Elevator".currentFloor, in2 := "Elevator".targetFloor)
      wire#w1
      S_Coil( "MoveTimerIN" )
   END_RUNG
   RUNG wire#w1
      R_Coil( #floorsubtracted )
   END_RUNG
   // the same network as SCL:
   IF ("Elevator".state = "ES_MOVING_DOWN") AND #floorsubtracted AND ("Elevator".currentFloor <> "Elevator".targetFloor) THEN
       "MoveTimerIN" := TRUE;
       #floorsubtracted := FALSE;
   END_IF;
END_REGION

REGION Network 16
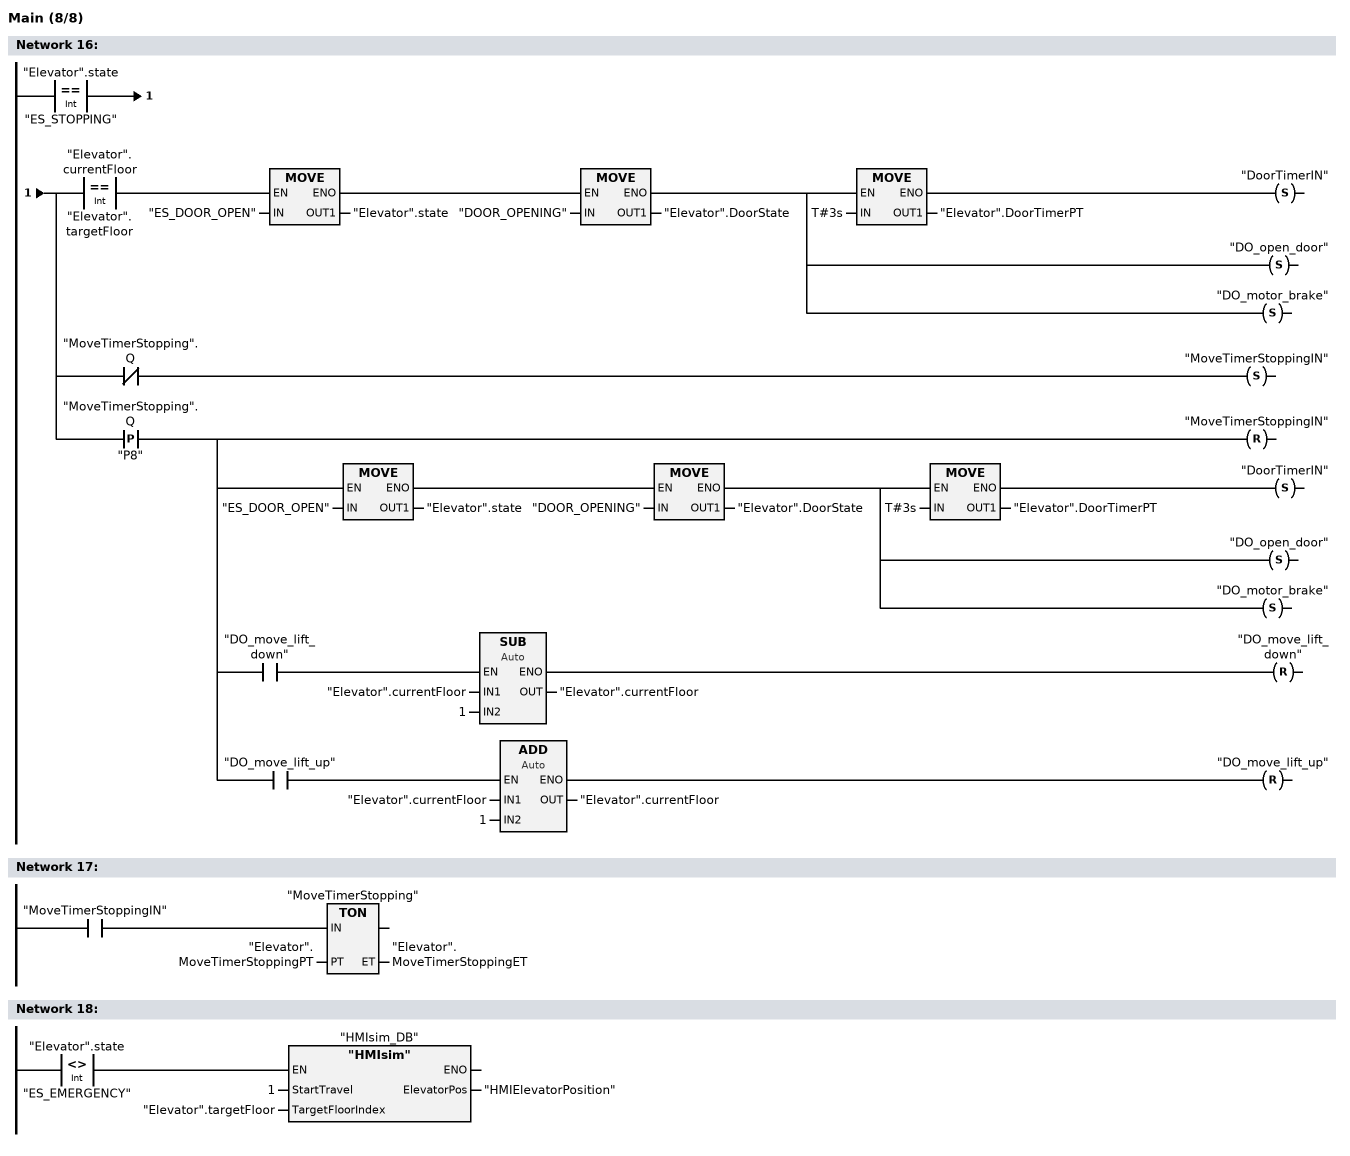
   RUNG wire#powerrail
      { S7_Templates := "SrcType := Int" } EQ_Contact(in1 := "Elevator".state, in2 := "ES_STOPPING")
      wire#w1
      { S7_Templates := "SrcType := Int" } EQ_Contact(in1 := "Elevator".currentFloor, in2 := "Elevator".targetFloor)
      { S7_GenerateENO := "TRUE" } Move(in := "ES_DOOR_OPEN", out1 => "Elevator".state)
      { S7_GenerateENO := "TRUE" } Move(in := "DOOR_OPENING", out1 => "Elevator".DoorState)
      wire#w2
      { S7_GenerateENO := "TRUE" } Move(in := T#3s, out1 => "Elevator".DoorTimerPT)
      S_Coil( "DoorTimerIN" )
   END_RUNG
   RUNG wire#w2
      S_Coil( "DO_open_door" )
   END_RUNG
   RUNG wire#w2
      S_Coil( "DO_motor_brake" )
   END_RUNG
   RUNG wire#w1
      I_Contact( "MoveTimerStopping".Q )
      S_Coil( "MoveTimerStoppingIN" )
   END_RUNG
   RUNG wire#w1
      P_Contact(operand := "MoveTimerStopping".Q, bit := "P8")
      wire#w3
      R_Coil( "MoveTimerStoppingIN" )
   END_RUNG
   RUNG wire#w3
      { S7_GenerateENO := "TRUE" } Move(in := "ES_DOOR_OPEN", out1 => "Elevator".state)
      { S7_GenerateENO := "TRUE" } Move(in := "DOOR_OPENING", out1 => "Elevator".DoorState)
      wire#w4
      { S7_GenerateENO := "TRUE" } Move(in := T#3s, out1 => "Elevator".DoorTimerPT)
      S_Coil( "DoorTimerIN" )
   END_RUNG
   RUNG wire#w4
      S_Coil( "DO_open_door" )
   END_RUNG
   RUNG wire#w4
      S_Coil( "DO_motor_brake" )
   END_RUNG
   RUNG wire#w3
      Contact( "DO_move_lift_down" )
      { S7_GenerateENO := "TRUE" } Sub(in1 := "Elevator".currentFloor, in2 := 1, out => "Elevator".currentFloor)
      R_Coil( "DO_move_lift_down" )
   END_RUNG
   RUNG wire#w3
      Contact( "DO_move_lift_up" )
      { S7_GenerateENO := "TRUE" } Add(in1 := "Elevator".currentFloor, in2 := 1, out => "Elevator".currentFloor)
      R_Coil( "DO_move_lift_up" )
   END_RUNG
   // the same network as SCL:
   // ENO of a box is taken as its EN; it also drops when the box reports an error
   #_w1 := "Elevator".state = "ES_STOPPING";
   IF #_w1 AND ("Elevator".currentFloor = "Elevator".targetFloor) THEN
       "Elevator".state := "ES_DOOR_OPEN";
       "Elevator".DoorState := "DOOR_OPENING";
       "Elevator".DoorTimerPT := T#3s;
       "DoorTimerIN" := TRUE;
       "DO_open_door" := TRUE;
       "DO_motor_brake" := TRUE;
   END_IF;
   IF #_w1 AND NOT "MoveTimerStopping".Q THEN "MoveTimerStoppingIN" := TRUE; END_IF;
   #_w2 := #_w1 AND "MoveTimerStopping".Q AND NOT "P8";   // rising edge of "MoveTimerStopping".Q
   "P8" := "MoveTimerStopping".Q;
   IF #_w2 THEN
       "MoveTimerStoppingIN" := FALSE;
       "Elevator".state := "ES_DOOR_OPEN";
       "Elevator".DoorState := "DOOR_OPENING";
       "Elevator".DoorTimerPT := T#3s;
       "DoorTimerIN" := TRUE;
       "DO_open_door" := TRUE;
       "DO_motor_brake" := TRUE;
   END_IF;
   IF #_w2 AND "DO_move_lift_down" THEN
       "Elevator".currentFloor := "Elevator".currentFloor - 1;
       "DO_move_lift_down" := FALSE;
   END_IF;
   IF #_w2 AND "DO_move_lift_up" THEN
       "Elevator".currentFloor := "Elevator".currentFloor + 1;
       "DO_move_lift_up" := FALSE;
   END_IF;
END_REGION

REGION Network 17
   "MoveTimerStopping".TON(IN := "MoveTimerStoppingIN",
                           PT := "Elevator".MoveTimerStoppingPT,
                           ET => "Elevator".MoveTimerStoppingET);
END_REGION

REGION Network 18
   RUNG wire#powerrail
      { S7_Templates := "SrcType := Int" } NE_Contact(in1 := "Elevator".state, in2 := "ES_EMERGENCY")
      "HMIsim_DB"(StartTravel := 1, TargetFloorIndex := "Elevator".targetFloor, ElevatorPos => "HMIElevatorPosition")
   END_RUNG
   // the same network as SCL:
   IF "Elevator".state <> "ES_EMERGENCY" THEN
       "HMIsim_DB"(StartTravel := 1,   // "HMIsim"
                   TargetFloorIndex := "Elevator".targetFloor,
                   ElevatorPos => "HMIElevatorPosition");
   END_IF;
END_REGION
END_ORGANIZATION_BLOCK

(* ===== HMI "HMI_RT_1" =====
system functions are stored by id; their names below are inferred from use
connection "HMI_Connection_2": ETHERNET, SMART_S7_1200_OMS

HMI tags "Default tag table"
   "Btn_0_floor_in" : Bool = PLC Btn_0_floor_in AT %M1.3, 1 s
   "Btn_1_floor_in" : Bool = PLC Btn_1_floor_in AT %M1.4, 1 s
   "Btn_10_floor_in" : Bool = PLC Btn_10_floor_in AT %M2.5, 1 s
   "Btn_2_floor_in" : Bool = PLC Btn_2_floor_in AT %M1.5, 1 s
   "Btn_3_floor_in" : Bool = PLC Btn_3_floor_in AT %M1.6, 1 s
   "Btn_4_floor_in" : Bool = PLC Btn_4_floor_in AT %M1.7, 1 s
   "Btn_5_floor_in" : Bool = PLC Btn_5_floor_in AT %M2.0, 1 s
   "Btn_6_floor_in" : Bool = PLC Btn_6_floor_in AT %M2.1, 1 s
   "Btn_7_floor_in" : Bool = PLC Btn_7_floor_in AT %M2.2, 1 s
   "Btn_8_floor_in" : Bool = PLC Btn_8_floor_in AT %M2.3, 1 s
   "Btn_9_floor_in" : Bool = PLC Btn_9_floor_in AT %M2.4, 1 s
   "HMIElevatorPosition" : Int = PLC HMIElevatorPosition AT %MW7, 1 s
   "Tag_ScreenNumber" : UInt, internal
   "Btn_emergency" : Bool = PLC Btn_emergency AT %M2.6, 1 s
   "Btn_close_door" : Bool = PLC Btn_close_door AT %M3.0, 1 s
   "Btn_open_door" : Bool = PLC Btn_open_door AT %M2.7, 1 s
   "HMIReq_0" : Bool = PLC HMIReq_0 AT %M4.1, 1 s
   "Btn_0_floor_out" : Bool = PLC Btn_0_floor_out AT %M0.0, 1 s
   "HMIReq_1" : Bool = PLC HMIReq_1 AT %M4.2, 1 s
   "HMIReq_2" : Bool = PLC HMIReq_2 AT %M4.3, 1 s
   "HMIReq_3" : Bool = PLC HMIReq_3 AT %M4.4, 1 s
   "HMIReq_4" : Bool = PLC HMIReq_4 AT %M4.5, 1 s
   "HMIReq_5" : Bool = PLC HMIReq_5 AT %M4.6, 1 s
   "HMIReq_6" : Bool = PLC HMIReq_6 AT %M4.7, 1 s
   "HMIReq_7" : Bool = PLC HMIReq_7 AT %M5.0, 1 s
   "HMIReq_8" : Bool = PLC HMIReq_8 AT %M5.1, 1 s
   "HMIReq_9" : Bool = PLC HMIReq_9 AT %M5.2, 1 s
   "HMIReq_10" : Bool = PLC HMIReq_10 AT %M5.3, 1 s
   "Btn_10_floor_out" : Bool = PLC Btn_10_floor_out AT %M1.2, 1 s
   "Btn_9_floor_out" : Bool = PLC Btn_9_floor_out AT %M1.1, 1 s
   "Btn_8_floor_out" : Bool = PLC Btn_8_floor_out AT %M1.0, 1 s
   "Btn_7_floor_out" : Bool = PLC Btn_7_floor_out AT %M0.7, 1 s
   "Btn_6_floor_out" : Bool = PLC Btn_6_floor_out AT %M0.6, 1 s
   "Btn_5_floor_out" : Bool = PLC Btn_5_floor_out AT %M0.5, 1 s
   "Btn_4_floor_out" : Bool = PLC Btn_4_floor_out AT %M0.4, 1 s
   "Btn_3_floor_out" : Bool = PLC Btn_3_floor_out AT %M0.3, 1 s
   "Btn_2_floor_out" : Bool = PLC Btn_2_floor_out AT %M0.2, 1 s
   "Btn_1_floor_out" : Bool = PLC Btn_1_floor_out AT %M0.1, 1 s
   "DO_move_lift_up" : Bool = PLC DO_move_lift_up AT %M3.3, 1 s
   "DO_move_lift_down" : Bool = PLC DO_move_lift_down AT %M3.4, 1 s
   "DO_open_door" : Bool = PLC DO_open_door AT %M3.1, 1 s
   "DO_close_door" : Bool = PLC DO_close_door AT %M3.2, 1 s
   "DO_motor_brake" : Bool = PLC DO_motor_brake AT %M3.5, 1 s

screen "Screen_1" 320x240
   Button "Button_1" at 270,97 size 25x32; TextOn '9'; TextOff '9'
      on Release: ResetBit("Btn_9_floor_in")
      on Press: SetBit("Btn_9_floor_in")
   Button "Button_2" at 195,54 size 25x32; TextOn '4'; TextOff '4'
      on Release: ResetBit("Btn_4_floor_in")
      on Press: SetBit("Btn_4_floor_in")
   Button "Button_3" at 233,54 size 25x32; TextOn '5'; TextOff '5'
      on Release: ResetBit("Btn_5_floor_in")
      on Press: SetBit("Btn_5_floor_in")
   Button "Button_4" at 270,54 size 25x32; TextOn '6'; TextOff '6'
      on Release: ResetBit("Btn_6_floor_in")
      on Press: SetBit("Btn_6_floor_in")
   Button "Button_5" at 195,11 size 25x32; TextOn '1'; TextOff '1'
      on Release: ResetBit("Btn_1_floor_in")
      on Press: SetBit("Btn_1_floor_in")
   Button "Button_6" at 270,11 size 25x32; TextOn '3'; TextOff '3'
      on Release: ResetBit("Btn_3_floor_in")
      on Press: SetBit("Btn_3_floor_in")
   Button "Button_7" at 233,11 size 25x32; TextOn '2'; TextOff '2'
      on Release: ResetBit("Btn_2_floor_in")
      on Press: SetBit("Btn_2_floor_in")
   Button "Button_8" at 195,142 size 25x32; TextOn '0'; TextOff '0'
      on Release: ResetBit("Btn_0_floor_in")
      on Press: SetBit("Btn_0_floor_in")
   Button "Button_9" at 195,97 size 25x32; TextOn '7'; TextOff '7'
      on Release: ResetBit("Btn_7_floor_in")
      on Press: SetBit("Btn_7_floor_in")
   Button "Button_10" at 233,97 size 25x32; TextOn '8'; TextOff '8'
      on Release: ResetBit("Btn_8_floor_in")
      on Press: SetBit("Btn_8_floor_in")
   Button "Button_11" at 270,142 size 25x32; TextOn '10'; TextOff '10'
      on Release: ResetBit("Btn_10_floor_in")
      on Press: SetBit("Btn_10_floor_in")
   Button "Button_12" at 195,186 size 25x32; TextOff 'Text'; PictureOff "Zrzut ekranu 2025-05-13 151421"
      on Release: ResetBit("Btn_close_door")
      on Press: SetBit("Btn_close_door")
   Button "Button_13" at 270,186 size 25x32; TextOff 'Text'; PictureOff "strzałki"
      on Release: ResetBit("Btn_open_door")
      on Press: SetBit("Btn_open_door")
   Button "Button_14" at 233,142 size 25x32; TextOff 'Text'; PictureOff "Graphic_1"
      on Press: InvertBit("Btn_emergency")
   Button "Button_15" at 56,197 size 20x17; TextOn '1'; TextOff '1'
      on Release: ResetBit("Btn_1_floor_out")
      on Press: SetBit("Btn_1_floor_out")
      Appearance <- "HMIReq_1"
   Button "Button_16" at 56,218 size 20x17; TextOn '0'; TextOff '0'
      on Release: ResetBit("Btn_0_floor_out")
      on Press: SetBit("Btn_0_floor_out")
      Appearance <- "HMIReq_0"
   Button "Button_17" at 56,177 size 20x17; TextOn '2'; TextOff '2'
      on Release: ResetBit("Btn_2_floor_out")
      on Press: SetBit("Btn_2_floor_out")
      Appearance <- "HMIReq_2"
   Button "Button_18" at 56,156 size 20x17; TextOn '3'; TextOff '3'
      on Release: ResetBit("Btn_3_floor_out")
      on Press: SetBit("Btn_3_floor_out")
      Appearance <- "HMIReq_3"
   Button "Button_19" at 56,135 size 20x17; TextOn '4'; TextOff '4'
      on Release: ResetBit("Btn_4_floor_out")
      on Press: SetBit("Btn_4_floor_out")
      Appearance <- "HMIReq_4"
   Button "Button_20" at 56,114 size 20x17; TextOn '5'; TextOff '5'
      on Release: ResetBit("Btn_5_floor_out")
      on Press: SetBit("Btn_5_floor_out")
      Appearance <- "HMIReq_5"
   Button "Button_21" at 56,93 size 20x17; TextOn '6'; TextOff '6'
      on Release: ResetBit("Btn_6_floor_out")
      on Press: SetBit("Btn_6_floor_out")
      Appearance <- "HMIReq_6"
   Button "Button_22" at 56,72 size 20x17; TextOn '7'; TextOff '7'
      on Release: ResetBit("Btn_7_floor_out")
      on Press: SetBit("Btn_7_floor_out")
      Appearance <- "HMIReq_7"
   Button "Button_23" at 56,51 size 20x17; TextOn '8'; TextOff '8'
      on Release: ResetBit("Btn_8_floor_out")
      on Press: SetBit("Btn_8_floor_out")
      Appearance <- "HMIReq_8"
   Button "Button_24" at 56,29 size 20x17; TextOn '9'; TextOff '9'
      on Release: ResetBit("Btn_9_floor_out")
      on Press: SetBit("Btn_9_floor_out")
      Appearance <- "HMIReq_9"
   Button "Button_25" at 56,8 size 20x17; TextOn '10'; TextOff '10'
      on Release: ResetBit("Btn_10_floor_out")
      on Press: SetBit("Btn_10_floor_out")
      Appearance <- "HMIReq_10"
   Circle "Circle_1" at 118,36 size 18x18
      Appearance <- "DO_move_lift_up"
   TextField "Text field_1" at 77,18 size 103x15; Text 'Ruch w górę / Moving up / Nach oben bewegen'
   Circle "Circle_2" at 118,71 size 18x18
      Appearance <- "DO_move_lift_down"
   TextField "Text field_2" at 72,53 size 107x15; Text 'Ruch w dół / Moving down / Nach unten bewegen'
   Circle "Circle_3" at 118,107 size 18x18
      Appearance <- "DO_open_door"
   TextField "Text field_3" at 84,91 size 90x15; Text 'Otwieranie drzwi / Opening doors / Türen öffnen'
   Circle "Circle_4" at 118,142 size 18x18
      Appearance <- "DO_close_door"
   TextField "Text field_4" at 82,127 size 89x15; Text 'Zamykanie drzwi / Closing doors / Türen schließen'
   Circle "Circle_5" at 118,176 size 18x18
      Appearance <- "DO_motor_brake"
   TextField "Text field_5" at 80,161 size 94x15; Text 'Hamulec windy / Elevator brake / Fahrstuhl-Bremse'
   Group "Group" at 19,218 size 18x17
      VerticalMovement <- "HMIElevatorPosition"
   Rectangle "Rectangle_24" at 28,218 size 9x17
      HorizontalMovement <- "HMIDoorPosition"
   Rectangle "Rectangle_25" at 19,218 size 9x17
      HorizontalMovement <- "HMIDoorPosition"
*)